    // ----------------------------------------------------------------------
    // Recirculate_Wash1:
    //  - Recirculates Wash 1 solvent to improve cleaning efficiency.
    // ----------------------------------------------------------------------
    E_WashingState.Recirculate_Wash1:

        RecirculateWash1();

        IF bMovementComplete THEN
            eWashingState    := E_WashingState.Cleaning_Lines_W1;
            iStepCounter     := 0;
            bMovementComplete := FALSE;
        END_IF


    // ----------------------------------------------------------------------
    // Cleaning_Lines_W1:
    //  - Cleans lines used for Wash 1 solvent.
    // ----------------------------------------------------------------------
    E_WashingState.Cleaning_Lines_W1:

        CleaningLinesWash1();

        IF bMovementComplete THEN
            eWashingState    := E_WashingState.Waste_Wash1;
            iStepCounter     := 0;
            bMovementComplete := FALSE;
        END_IF


    // ----------------------------------------------------------------------
    // Waste_Wash1:
    //  - Sends Wash 1 solvent remaining in lines to waste.
    //  - Then decides whether Wash 2 is enabled by recipe.
    // ----------------------------------------------------------------------
    E_WashingState.Waste_Wash1:

        WasteWash1();

        IF bMovementComplete THEN
            iStepCounter     := 0;
            bMovementComplete := FALSE;

            // Check if Wash 2 is active in the recipe:
            // aSolventN[4] > 0 → Wash 2 enabled
            IF GVL_Recipe.stActiveRecipe.stSolventsTimes.aSolventN[4] > 0 THEN
                eWashingState := E_WashingState.Metering_Wash2;
            ELSE
                eWashingState := E_WashingState.Completed;
            END_IF
        END_IF


    // ----------------------------------------------------------------------
    // Metering_Wash2:
    //  - Meters solvent for Wash 2 if configured in recipe.
    // ----------------------------------------------------------------------
    E_WashingState.Metering_Wash2:

        MeteringWash2();

        IF bMovementComplete THEN
            eWashingState    := E_WashingState.Recirculate_Wash2;
            iStepCounter     := 0;
            bMovementComplete := FALSE;
        END_IF


    // ----------------------------------------------------------------------
    // Recirculate_Wash2:
    //  - Recirculates Wash 2 solvent.
    // ----------------------------------------------------------------------
    E_WashingState.Recirculate_Wash2:

        RecirculateWash2();

        IF bMovementComplete THEN
            eWashingState    := E_WashingState.Cleaning_Lines_W2;
            iStepCounter     := 0;
            bMovementComplete := FALSE;
        END_IF


    // ----------------------------------------------------------------------
    // Cleaning_Lines_W2:
    //  - Cleans lines used for Wash 2 solvent.
    // ----------------------------------------------------------------------
    E_WashingState.Cleaning_Lines_W2:

        CleaningLinesWash2();

        IF bMovementComplete THEN
            eWashingState    := E_WashingState.Waste_Wash2;
            iStepCounter     := 0;
            bMovementComplete := FALSE;
        END_IF


    // ----------------------------------------------------------------------
    // Waste_Wash2:
    //  - Sends Wash 2 solvent remaining in lines to waste.
    // ----------------------------------------------------------------------
    E_WashingState.Waste_Wash2:

        WasteWash2();

        IF bMovementComplete THEN
            iStepCounter     := 0;
            bMovementComplete := FALSE;
            eWashingState    := E_WashingState.Completed;
        END_IF


    // ----------------------------------------------------------------------
    // Completed:
    //  - Washing phase has finished successfully.
    //  - Updates HMI and raises bWashingDone.
    // ----------------------------------------------------------------------
    E_WashingState.Completed:

        GVL_HMI.HMIAnimation.sLoadTextWashing   := 'Completed';
        GVL_HMI.HMIAnimation.rLoadBarWashing    := 100.0;
        GVL_HMI.HMIAnimation.eIconStateWashing  := E_IconState.Completed;

        bWashingDone  := TRUE;
        bWashingError := FALSE;


    // ----------------------------------------------------------------------
    // Error:
    //  - Generic washing error state (hook for future error handling).
    //  - Currently sets HMI to "Error" and raises bWashingError.
    // ----------------------------------------------------------------------
    E_WashingState.Error:

        GVL_HMI.HMIAnimation.sLoadTextWashing   := 'Error';
        GVL_HMI.HMIAnimation.rLoadBarWashing    := 0.0;
        GVL_HMI.HMIAnimation.eIconStateWashing  := E_IconState.Waiting;

        bWashingError := TRUE;
        bWashingDone  := FALSE;

END_CASE

ACTION CleaningLinesWash1:
//Exactly the oppisite of Recirculate Wash 1
CASE iStepCounter OF
	
	0: //Provide HMI animation details
		GVL_HMI.HMIAnimation.sLoadTextWashing := 'Cleaning Lines W1'; 
		iStepCounter := 1;
		
		FOR i := 1 TO 5 DO
			bMoveValveDone[i] := FALSE;
		END_FOR
		
    1: // Set valves on position 5 (Recirculating)
    	FOR i := 1 TO 5 DO
			IF NOT bMoveValveDone[i] THEN
			bMoveValveDone[i] := GVL_Motion.aValvesObj[i].MoveValve( iPosition := 5, 
																	 rVelocity := GVL_Motion.aValves[i].rTargetVel, 
																	 rAcc := GVL_Motion.aValves[i].rAcceleration, 
																	 rDec := GVL_Motion.aValves[i].rDeceleration 
																	);
			END_IF
		END_FOR
		
		IF bMoveValveDone[1] AND bMoveValveDone[2] AND bMoveValveDone[3] AND bMoveValveDone[4] AND bMoveValveDone[5] THEN
			FOR i := 1 TO 5 DO
				bMoveValveDone[i] := FALSE;
        	END_FOR
        	iStepCounter := 2;
		END_IF

    2: // Calculates the number of degrees of rotation of the pumps based on Wash 1 volume and factor 2

		fDistance[1] := F_VolumeToSteps(rVolume := (GVL_Recipe.stActiveRecipe.stVolumes.aT_IC_Volume[3] + GVL_Motion.aPumps[1].Rotary.rDeadVolume) * 2, iPumpIndex := 1);
		fDistance[2] := F_VolumeToSteps(rVolume := (GVL_Recipe.stActiveRecipe.stVolumes.aS0_Volume[3] + GVL_Motion.aPumps[2].Rotary.rDeadVolume) * 2, iPumpIndex := 2);
		fDistance[3] := F_VolumeToSteps(rVolume := (GVL_Recipe.stActiveRecipe.stVolumes.aS1_Volume[3] + GVL_Motion.aPumps[3].Rotary.rDeadVolume) * 2, iPumpIndex := 3);
		fDistance[4] := F_VolumeToSteps(rVolume := (GVL_Recipe.stActiveRecipe.stVolumes.aS2_Volume[3] + GVL_Motion.aPumps[4].Rotary.rDeadVolume) * 2, iPumpIndex := 4);
		fDistance[5] := F_VolumeToSteps(rVolume := (GVL_Recipe.stActiveRecipe.stVolumes.aS3_Volume[3] + GVL_Motion.aPumps[5].Rotary.rDeadVolume) * 2, iPumpIndex := 5);
		fDistance[6] := F_VolumeToSteps(rVolume := (GVL_Recipe.stActiveRecipe.stVolumes.aS4_Volume[3] + GVL_Motion.aPumps[6].Rotary.rDeadVolume) * 2, iPumpIndex := 6);
		fDistance[7] := F_VolumeToSteps(rVolume := (GVL_Recipe.stActiveRecipe.stVolumes.aS5_Volume[3] + GVL_Motion.aPumps[7].Rotary.rDeadVolume) * 2, iPumpIndex := 7);
		fDistance[8] := F_VolumeToSteps(rVolume := (GVL_Recipe.stActiveRecipe.stVolumes.aS6_Volume[3] + GVL_Motion.aPumps[8].Rotary.rDeadVolume) * 2, iPumpIndex := 8);
		fDistance[9] := F_VolumeToSteps(rVolume := (GVL_Recipe.stActiveRecipe.stVolumes.aS7_Volume[3] + GVL_Motion.aPumps[9].Rotary.rDeadVolume) * 2, iPumpIndex := 9);
		fDistance[10] := F_VolumeToSteps(rVolume := (GVL_Recipe.stActiveRecipe.stVolumes.aF_Volume[3] + GVL_Motion.aPumps[10].Rotary.rDeadVolume) * 2, iPumpIndex := 10);

		FOR i := 1 TO 10 DO
			bMovePumpDone[i] := FALSE;
		END_FOR
		
		iStepCounter := 3;
		
    3: // Starts rotary movement with calculated distance (degrees/sec -> steps) [positive movement]
        FOR i := 1 TO 10 DO
			IF NOT bMovePumpDone[i] THEN
				bMovePumpDone[i] := GVL_Motion.aPumpsRotary[i].MoveRelative( Distance := fDistance[i],
																			 Velocity := GVL_Settings.stPumpParameters.iRunVelocity * 6, 
																			 Acc := GVL_Settings.stPumpParameters.iRunVelocity * 3, 
																			 Dec := GVL_Settings.stPumpParameters.iRunVelocity * 3 
																			);
			END_IF
        END_FOR
		IF bMovePumpDone[1] AND bMovePumpDone[2] AND bMovePumpDone[3] AND bMovePumpDone[4] AND bMovePumpDone[5] AND bMovePumpDone[6] AND bMovePumpDone[7] AND bMovePumpDone[8] AND bMovePumpDone[9] AND bMovePumpDone[10] THEN
			FOR i := 1 TO 10 DO
				bMovePumpDone[i] := FALSE;
        	END_FOR
        	iStepCounter := 4; // Move to next step
		END_IF

    4: // Sets the movement done flag
		bMovementComplete := TRUE;
	
        
END_CASE
END_ACTION

ACTION CleaningLinesWash2:
//Exactly the oppisite of Recirculate Wash 1
CASE iStepCounter OF
	
	0: //Provide HMI animation details
		GVL_HMI.HMIAnimation.sLoadTextWashing := 'Cleaning Lines W2'; 
		iStepCounter := 1;
		
		FOR i := 1 TO 5 DO
			bMoveValveDone[i] := FALSE;
		END_FOR
		
    1: // Set valves on position 5 (Recirculating)
    	FOR i := 1 TO 5 DO
			IF NOT bMoveValveDone[i] THEN
			bMoveValveDone[i] := GVL_Motion.aValvesObj[i].MoveValve( iPosition := 5, 
																	 rVelocity := GVL_Motion.aValves[i].rTargetVel, 
																	 rAcc := GVL_Motion.aValves[i].rAcceleration, 
																	 rDec := GVL_Motion.aValves[i].rDeceleration 
																	);
			END_IF
		END_FOR
		
		IF bMoveValveDone[1] AND bMoveValveDone[2] AND bMoveValveDone[3] AND bMoveValveDone[4] AND bMoveValveDone[5] THEN
			FOR i := 1 TO 5 DO
				bMoveValveDone[i] := FALSE;
        	END_FOR
        	iStepCounter := 2;
		END_IF

    2: //Calculates the number of degrees of rotation of the pumps based on Wash 2 volume and factor 2

    	fDistance[1] := F_VolumeToSteps(rVolume := (GVL_Recipe.stActiveRecipe.stVolumes.aT_IC_Volume[4] + GVL_Motion.aPumps[1].Rotary.rDeadVolume) * 2, iPumpIndex := 1);
		fDistance[2] := F_VolumeToSteps(rVolume := (GVL_Recipe.stActiveRecipe.stVolumes.aS0_Volume[4] + GVL_Motion.aPumps[2].Rotary.rDeadVolume) * 2, iPumpIndex := 2);
		fDistance[3] := F_VolumeToSteps(rVolume := (GVL_Recipe.stActiveRecipe.stVolumes.aS1_Volume[4] + GVL_Motion.aPumps[3].Rotary.rDeadVolume) * 2, iPumpIndex := 3);
		fDistance[4] := F_VolumeToSteps(rVolume := (GVL_Recipe.stActiveRecipe.stVolumes.aS2_Volume[4] + GVL_Motion.aPumps[4].Rotary.rDeadVolume) * 2, iPumpIndex := 4);
		fDistance[5] := F_VolumeToSteps(rVolume := (GVL_Recipe.stActiveRecipe.stVolumes.aS3_Volume[4] + GVL_Motion.aPumps[5].Rotary.rDeadVolume) * 2, iPumpIndex := 5);
		fDistance[6] := F_VolumeToSteps(rVolume := (GVL_Recipe.stActiveRecipe.stVolumes.aS4_Volume[4] + GVL_Motion.aPumps[6].Rotary.rDeadVolume) * 2, iPumpIndex := 6);
		fDistance[7] := F_VolumeToSteps(rVolume := (GVL_Recipe.stActiveRecipe.stVolumes.aS5_Volume[4] + GVL_Motion.aPumps[7].Rotary.rDeadVolume) * 2, iPumpIndex := 7);
		fDistance[8] := F_VolumeToSteps(rVolume := (GVL_Recipe.stActiveRecipe.stVolumes.aS6_Volume[4] + GVL_Motion.aPumps[8].Rotary.rDeadVolume) * 2, iPumpIndex := 8);
		fDistance[9] := F_VolumeToSteps(rVolume := (GVL_Recipe.stActiveRecipe.stVolumes.aS7_Volume[4] + GVL_Motion.aPumps[9].Rotary.rDeadVolume) * 2, iPumpIndex := 9);
		fDistance[10] := F_VolumeToSteps(rVolume := (GVL_Recipe.stActiveRecipe.stVolumes.aF_Volume[4] + GVL_Motion.aPumps[10].Rotary.rDeadVolume) * 2, iPumpIndex := 10);

		FOR i := 1 TO 10 DO
			bMovePumpDone[i] := FALSE;
		END_FOR
		
		iStepCounter := 3;
		
    3: // Starts rotary movement with calculated distance (degrees/sec -> steps) [positive movement]
        FOR i := 1 TO 10 DO
			IF NOT bMovePumpDone[i] THEN
				bMovePumpDone[i] := GVL_Motion.aPumpsRotary[i].MoveRelative( Distance := fDistance[i],
																			 Velocity := GVL_Settings.stPumpParameters.iRunVelocity * 6, 
																			 Acc := GVL_Settings.stPumpParameters.iRunVelocity * 3, 
																			 Dec := GVL_Settings.stPumpParameters.iRunVelocity * 3 
																			);
			END_IF
        END_FOR
		IF bMovePumpDone[1] AND bMovePumpDone[2] AND bMovePumpDone[3] AND bMovePumpDone[4] AND bMovePumpDone[5] AND bMovePumpDone[6] AND bMovePumpDone[7] AND bMovePumpDone[8] AND bMovePumpDone[9] AND bMovePumpDone[10] THEN
			FOR i := 1 TO 10 DO
				bMovePumpDone[i] := FALSE;
        	END_FOR
        	iStepCounter := 4; // Move to next step
		END_IF

    4: // Sets the movement done flag
		bMovementComplete := TRUE;
	
        
END_CASE
END_ACTION

METHOD EstimateTotalTime : REAL
VAR
	i : INT;
    rTotalTime : REAL := 0.0;
    rTmpTime : REAL;
    rMaxPumpTime : REAL;
	aVolumesW1 : ARRAY[1..10] OF REAL;
	aVolumesW2 : ARRAY[1..10] OF REAL;
	rM2Travel : lREAL;
END_VAR
// --- Valve movements ---
// Estimated 1s per group of 5 valves per change (6 changes)
rTotalTime := rTotalTime + 1 * 6;

// --- Motor M2 movements --- (used in WasteWash1 and WasteWash2)
rM2Travel :=  ABS(GVL_Settings.stMachineParam.aM2Position[2] - GVL_Settings.stMachineParam.aM2Position[1]) / GVL_Settings.stMachineParam.rM2Velocity  //Waste Position Move
			+ ABS(GVL_Settings.stMachineParam.aM2Position[2] - GVL_Settings.stMachineParam.aM2Position[1]) / GVL_Settings.stMachineParam.rM2Velocity; //Home Position Move

rTotalTime := rTotalTime + rM2Travel * 2;

// --- Agitations (Recirculations) ---
rTotalTime := rTotalTime + TO_REAL(GVL_Recipe.stActiveRecipe.stOtherParams.tAgitate1Time) / 1000.0;
rTotalTime := rTotalTime + TO_REAL(GVL_Recipe.stActiveRecipe.stOtherParams.tAgitate2Time) / 1000.0;

// --- Pump phases executed in parallel ---
//Volume value tranfer Wash 1
aVolumesW1[1] := GVL_Recipe.stActiveRecipe.stVolumes.aT_IC_Volume[3];
aVolumesW1[2] := GVL_Recipe.stActiveRecipe.stVolumes.aS0_Volume[3];
aVolumesW1[3] := GVL_Recipe.stActiveRecipe.stVolumes.aS1_Volume[3];
aVolumesW1[4] := GVL_Recipe.stActiveRecipe.stVolumes.aS2_Volume[3];
aVolumesW1[5] := GVL_Recipe.stActiveRecipe.stVolumes.aS3_Volume[3];
aVolumesW1[6] := GVL_Recipe.stActiveRecipe.stVolumes.aS4_Volume[3];
aVolumesW1[7] := GVL_Recipe.stActiveRecipe.stVolumes.aS5_Volume[3];
aVolumesW1[8] := GVL_Recipe.stActiveRecipe.stVolumes.aS6_Volume[3];
aVolumesW1[9] := GVL_Recipe.stActiveRecipe.stVolumes.aS7_Volume[3];
aVolumesW1[10] := GVL_Recipe.stActiveRecipe.stVolumes.aF_Volume[3];
//Volume value tranfer Wash 2
aVolumesW2[1] := GVL_Recipe.stActiveRecipe.stVolumes.aT_IC_Volume[4];
aVolumesW2[2] := GVL_Recipe.stActiveRecipe.stVolumes.aS0_Volume[4];
aVolumesW2[3] := GVL_Recipe.stActiveRecipe.stVolumes.aS1_Volume[4];
aVolumesW2[4] := GVL_Recipe.stActiveRecipe.stVolumes.aS2_Volume[4];
aVolumesW2[5] := GVL_Recipe.stActiveRecipe.stVolumes.aS3_Volume[4];
aVolumesW2[6] := GVL_Recipe.stActiveRecipe.stVolumes.aS4_Volume[4];
aVolumesW2[7] := GVL_Recipe.stActiveRecipe.stVolumes.aS5_Volume[4];
aVolumesW2[8] := GVL_Recipe.stActiveRecipe.stVolumes.aS6_Volume[4];
aVolumesW2[9] := GVL_Recipe.stActiveRecipe.stVolumes.aS7_Volume[4];
aVolumesW2[10] := GVL_Recipe.stActiveRecipe.stVolumes.aF_Volume[4];

// For each block, use only the slowest pump
// MeteringWash1 (SolventN[3], Volumes[i][3])
IF GVL_Recipe.stActiveRecipe.stSolventsTimes.aSolventN[3] > 0 THEN
	rMaxPumpTime := 0;
	FOR i := 1 TO 10 DO
		rTmpTime := F_VolumeToSteps(rVolume := aVolumesW1[i], iPumpIndex := i) / GVL_Motion.aPumps[i].Rotary.rSpeed;
		IF rTmpTime > rMaxPumpTime THEN rMaxPumpTime := rTmpTime; END_IF
	END_FOR
	rTotalTime := rTotalTime + rMaxPumpTime;
END_IF

// MeteringWash2 (SolventN[4], Volumes[i][4])
IF GVL_Recipe.stActiveRecipe.stSolventsTimes.aSolventN[4] > 0 THEN
	rMaxPumpTime := 0;
	FOR i := 1 TO 10 DO
		rTmpTime := F_VolumeToSteps(rVolume := aVolumesW2[i], iPumpIndex := i) / GVL_Motion.aPumps[i].Rotary.rSpeed;
		IF rTmpTime > rMaxPumpTime THEN rMaxPumpTime := rTmpTime; END_IF
	END_FOR
	rTotalTime := rTotalTime + rMaxPumpTime;
END_IF

// WasteWash1 includes recipe volume + tubing dead volume (for each pump)
IF GVL_Recipe.stActiveRecipe.stSolventsTimes.aSolventN[3] > 0 THEN
	rMaxPumpTime := 0;
	FOR i := 1 TO 10 DO
		rTmpTime := F_VolumeToSteps(rVolume := aVolumesW1[i] + GVL_Motion.aPumps[i].Rotary.rDeadVolume, iPumpIndex := i) / GVL_Motion.aPumps[i].Rotary.rSpeed;
		IF rTmpTime > rMaxPumpTime THEN rMaxPumpTime := rTmpTime; END_IF
	END_FOR
	rTotalTime := rTotalTime + rMaxPumpTime;
END_IF

// WasteWash2 includes recipe volume + tubing dead volume (for each pump)
IF GVL_Recipe.stActiveRecipe.stSolventsTimes.aSolventN[4] > 0 THEN
	rMaxPumpTime := 0;
	FOR i := 1 TO 10 DO
		rTmpTime := F_VolumeToSteps(rVolume := aVolumesW2[i] + GVL_Motion.aPumps[i].Rotary.rDeadVolume, iPumpIndex := i) / GVL_Motion.aPumps[i].Rotary.rSpeed;
		IF rTmpTime > rMaxPumpTime THEN rMaxPumpTime := rTmpTime; END_IF
	END_FOR
	rTotalTime := rTotalTime + rMaxPumpTime;
END_IF

EstimateTotalTime := rTotalTime;
END_METHOD

ACTION MeteringWash1:
CASE iStepCounter OF
	
	0: //Provide HMI animation details
		GVL_HMI.HMIAnimation.sLoadTextWashing := 'Metering Wash 1'; 
		iStepCounter := 1; 
		FOR i := 1 TO 5 DO //reset valve movement flags
			bMoveValveDone[i] := FALSE;
		END_FOR
		
    1: // Set valves for Wash 1 position
	    FOR i := 1 TO 5 DO
			IF NOT bMoveValveDone[i] THEN
				bMoveValveDone[i] := GVL_Motion.aValvesObj[i].MoveValve(iPosition := GVL_Recipe.stActiveRecipe.stSolventsTimes.aSolventN[3], //Wash 1 solvent position
																	 	rVelocity := GVL_Motion.aValves[i].rTargetVel, 
																	 	rAcc := GVL_Motion.aValves[i].rAcceleration, 
																	 	rDec := GVL_Motion.aValves[i].rDeceleration 
																		);
			END_IF
			
        END_FOR
		
		IF bMoveValveDone[1] AND bMoveValveDone[2] AND bMoveValveDone[3] AND bMoveValveDone[4] AND bMoveValveDone[5] THEN
			FOR i := 1 TO 5 DO
				bMoveValveDone[i] := FALSE;
        	END_FOR
        	iStepCounter := 2;
		END_IF
        
	2: //Calculating the distance for each pump based on recipe volume plus tubing dead volume [Wash 1 - index 3]
		fDistance[1] := F_VolumeToSteps(rVolume := GVL_Recipe.stActiveRecipe.stVolumes.aT_IC_Volume[3] + GVL_Motion.aPumps[1].Rotary.rDeadVolume, iPumpIndex := 1);
		fDistance[2] := F_VolumeToSteps(rVolume := GVL_Recipe.stActiveRecipe.stVolumes.aS0_Volume[3] + GVL_Motion.aPumps[2].Rotary.rDeadVolume, iPumpIndex := 2);
		fDistance[3] := F_VolumeToSteps(rVolume := GVL_Recipe.stActiveRecipe.stVolumes.aS1_Volume[3] + GVL_Motion.aPumps[3].Rotary.rDeadVolume, iPumpIndex := 3);
		fDistance[4] := F_VolumeToSteps(rVolume := GVL_Recipe.stActiveRecipe.stVolumes.aS2_Volume[3] + GVL_Motion.aPumps[4].Rotary.rDeadVolume, iPumpIndex := 4);
		fDistance[5] := F_VolumeToSteps(rVolume := GVL_Recipe.stActiveRecipe.stVolumes.aS3_Volume[3] + GVL_Motion.aPumps[5].Rotary.rDeadVolume, iPumpIndex := 5);
		fDistance[6] := F_VolumeToSteps(rVolume := GVL_Recipe.stActiveRecipe.stVolumes.aS4_Volume[3] + GVL_Motion.aPumps[6].Rotary.rDeadVolume, iPumpIndex := 6);
		fDistance[7] := F_VolumeToSteps(rVolume := GVL_Recipe.stActiveRecipe.stVolumes.aS5_Volume[3] + GVL_Motion.aPumps[7].Rotary.rDeadVolume, iPumpIndex := 7);
		fDistance[8] := F_VolumeToSteps(rVolume := GVL_Recipe.stActiveRecipe.stVolumes.aS6_Volume[3] + GVL_Motion.aPumps[8].Rotary.rDeadVolume, iPumpIndex := 8);
		fDistance[9] := F_VolumeToSteps(rVolume := GVL_Recipe.stActiveRecipe.stVolumes.aS7_Volume[3] + GVL_Motion.aPumps[9].Rotary.rDeadVolume, iPumpIndex := 9);
		fDistance[10] := F_VolumeToSteps(rVolume := GVL_Recipe.stActiveRecipe.stVolumes.aF_Volume[3] + GVL_Motion.aPumps[10].Rotary.rDeadVolume, iPumpIndex := 10);
		
		FOR i := 1 TO 10 DO //reset pump movement flags
			bMovePumpDone[i] := FALSE;
		END_FOR
		
		iStepCounter := 3;
		
    3: // Performs rotary movement (positive movement)
        FOR i := 1 TO 10 DO
            IF NOT bMovePumpDone[i] THEN
				bMovePumpDone[i] := GVL_Motion.aPumpsRotary[i].MoveRelative( Distance := fDistance[i],
																			 Velocity := GVL_Settings.stPumpParameters.iMeterVelocity * 6,
																			 Acc := GVL_Settings.stPumpParameters.iMeterVelocity * 3, 
																			 Dec := GVL_Settings.stPumpParameters.iMeterVelocity * 3 
																			);
			END_IF
        END_FOR
		IF bMovePumpDone[1] AND bMovePumpDone[2] AND bMovePumpDone[3] AND bMovePumpDone[4] AND bMovePumpDone[5] AND bMovePumpDone[6] AND bMovePumpDone[7] AND bMovePumpDone[8] AND bMovePumpDone[9] AND bMovePumpDone[10] THEN
			FOR i := 1 TO 10 DO
				bMovePumpDone[i] := FALSE;
        	END_FOR
        	iStepCounter := 4; // Move to next step to monitor completion
		END_IF
	
	4: // Sets the movement done flag
		bMovementComplete := TRUE;
         
END_CASE
END_ACTION

ACTION MeteringWash2:
CASE iStepCounter OF
	
	0: //Provide HMI animation details
		GVL_HMI.HMIAnimation.sLoadTextWashing := 'Metering Wash 2'; 
		iStepCounter := 1; 
		FOR i := 1 TO 5 DO //reset valve movement flags
			bMoveValveDone[i] := FALSE;
		END_FOR
		
    1: // Set valves for Rinse 1 position
	    FOR i := 1 TO 5 DO
			IF NOT bMoveValveDone[i] THEN
				bMoveValveDone[i] := GVL_Motion.aValvesObj[i].MoveValve(iPosition := GVL_Recipe.stActiveRecipe.stSolventsTimes.aSolventN[4], //Wash 2 solvent position
																	 	rVelocity := GVL_Motion.aValves[i].rTargetVel, 
																	 	rAcc := GVL_Motion.aValves[i].rAcceleration, 
																	 	rDec := GVL_Motion.aValves[i].rDeceleration 
																		);
			END_IF
			
        END_FOR
		
		IF bMoveValveDone[1] AND bMoveValveDone[2] AND bMoveValveDone[3] AND bMoveValveDone[4] AND bMoveValveDone[5] THEN
			FOR i := 1 TO 5 DO
				bMoveValveDone[i] := FALSE;
        	END_FOR
        	iStepCounter := 2;
		END_IF
        
	2: //Calculating the distance for each pump based on recipe volume plus tubing dead volume [Wash 2 - index 4]
		fDistance[1] := F_VolumeToSteps(rVolume := GVL_Recipe.stActiveRecipe.stVolumes.aT_IC_Volume[4] + GVL_Motion.aPumps[1].Rotary.rDeadVolume, iPumpIndex := 1);
		fDistance[2] := F_VolumeToSteps(rVolume := GVL_Recipe.stActiveRecipe.stVolumes.aS0_Volume[4] + GVL_Motion.aPumps[2].Rotary.rDeadVolume, iPumpIndex := 2);
		fDistance[3] := F_VolumeToSteps(rVolume := GVL_Recipe.stActiveRecipe.stVolumes.aS1_Volume[4] + GVL_Motion.aPumps[3].Rotary.rDeadVolume, iPumpIndex := 3);
		fDistance[4] := F_VolumeToSteps(rVolume := GVL_Recipe.stActiveRecipe.stVolumes.aS2_Volume[4] + GVL_Motion.aPumps[4].Rotary.rDeadVolume, iPumpIndex := 4);
		fDistance[5] := F_VolumeToSteps(rVolume := GVL_Recipe.stActiveRecipe.stVolumes.aS3_Volume[4] + GVL_Motion.aPumps[5].Rotary.rDeadVolume, iPumpIndex := 5);
		fDistance[6] := F_VolumeToSteps(rVolume := GVL_Recipe.stActiveRecipe.stVolumes.aS4_Volume[4] + GVL_Motion.aPumps[6].Rotary.rDeadVolume, iPumpIndex := 6);
		fDistance[7] := F_VolumeToSteps(rVolume := GVL_Recipe.stActiveRecipe.stVolumes.aS5_Volume[4] + GVL_Motion.aPumps[7].Rotary.rDeadVolume, iPumpIndex := 7);
		fDistance[8] := F_VolumeToSteps(rVolume := GVL_Recipe.stActiveRecipe.stVolumes.aS6_Volume[4] + GVL_Motion.aPumps[8].Rotary.rDeadVolume, iPumpIndex := 8);
		fDistance[9] := F_VolumeToSteps(rVolume := GVL_Recipe.stActiveRecipe.stVolumes.aS7_Volume[4] + GVL_Motion.aPumps[9].Rotary.rDeadVolume, iPumpIndex := 9);
		fDistance[10] := F_VolumeToSteps(rVolume := GVL_Recipe.stActiveRecipe.stVolumes.aF_Volume[4] + GVL_Motion.aPumps[10].Rotary.rDeadVolume, iPumpIndex := 10);
		
		FOR i := 1 TO 10 DO //reset pump movement flags
			bMovePumpDone[i] := FALSE;
		END_FOR
		
		iStepCounter := 3;
		
    3: // Performs rotary movement (positive movement)
        FOR i := 1 TO 10 DO
            IF NOT bMovePumpDone[i] THEN
				bMovePumpDone[i] := GVL_Motion.aPumpsRotary[i].MoveRelative( Distance := fDistance[i],
																			 Velocity := GVL_Settings.stPumpParameters.iMeterVelocity * 6,
																			 Acc := GVL_Settings.stPumpParameters.iMeterVelocity * 3, 
																			 Dec := GVL_Settings.stPumpParameters.iMeterVelocity * 3 
																			);
			END_IF
        END_FOR
		IF bMovePumpDone[1] AND bMovePumpDone[2] AND bMovePumpDone[3] AND bMovePumpDone[4] AND bMovePumpDone[5] AND bMovePumpDone[6] AND bMovePumpDone[7] AND bMovePumpDone[8] AND bMovePumpDone[9] AND bMovePumpDone[10] THEN
			FOR i := 1 TO 10 DO
				bMovePumpDone[i] := FALSE;
        	END_FOR
        	iStepCounter := 4; // Move to next step to monitor completion
		END_IF
	
	4: // Sets the movement done flag
		bMovementComplete := TRUE;
         
END_CASE
END_ACTION

ACTION RecirculateWash1:
CASE iStepCounter OF
	
	0: //Provide HMI animation details
		GVL_HMI.HMIAnimation.sLoadTextWashing := 'Recirculate Wash 1'; 
		FOR i := 1 TO 5 DO
			bMoveValveDone[i] := FALSE;
		END_FOR
		iStepCounter := 1;
		
    1: // Set Valves position 5 (Recirculate)
    	FOR i := 1 TO 5 DO
			IF NOT bMoveValveDone[i] THEN
			bMoveValveDone[i] := GVL_Motion.aValvesObj[i].MoveValve( iPosition := 5, 
																	 rVelocity := GVL_Motion.aValves[i].rTargetVel, 
																	 rAcc := GVL_Motion.aValves[i].rAcceleration, 
																	 rDec := GVL_Motion.aValves[i].rDeceleration 
																	);
			END_IF
		END_FOR
		
		IF bMoveValveDone[1] AND bMoveValveDone[2] AND bMoveValveDone[3] AND bMoveValveDone[4] AND bMoveValveDone[5] THEN
			FOR i := 1 TO 5 DO
				bMoveValveDone[i] := FALSE;
        	END_FOR
        	iStepCounter := 2;
		END_IF

    2: // Calcula o numero de graus de rotacao das bombas baseado no tempo da receita Agitate Time 1

		fRecirculationTime  := TO_REAL(TIME_TO_DWORD(GVL_Recipe.stCurrentRecipe.stSolventsTimes.aTime[3])/1000);
		FOR i := 1 TO 10 DO
			fCalcDistance[i] 	:= fRecirculationTime * (GVL_Recipe.stActiveRecipe.stSolventsTimes.aVelocity[3] * 6);
		END_FOR
		
		FOR i := 1 TO 10 DO
			bMovePumpDone[i] := FALSE;
		END_FOR
		
		IF fRecirculationTime > 0 THEN
			iStepCounter := 3;
		END_IF
		
    3: // Inicia movimento rotativo com distância calculada (graus/seg -> steps) [negative moviment]
        FOR i := 1 TO 10 DO
			IF NOT bMovePumpDone[i] THEN
				bMovePumpDone[i] := GVL_Motion.aPumpsRotary[i].MoveRelative( Distance := - fCalcDistance[i],
																			 Velocity := GVL_Recipe.stActiveRecipe.stSolventsTimes.aVelocity[3] * 6, 
																			 Acc := GVL_Recipe.stActiveRecipe.stSolventsTimes.aVelocity[3] * 6, 
																			 Dec := GVL_Recipe.stActiveRecipe.stSolventsTimes.aVelocity[3] * 6 
																			);
			END_IF
        END_FOR
		IF bMovePumpDone[1] AND bMovePumpDone[2] AND bMovePumpDone[3] AND bMovePumpDone[4] AND bMovePumpDone[5] AND bMovePumpDone[6] AND bMovePumpDone[7] AND bMovePumpDone[8] AND bMovePumpDone[9] AND bMovePumpDone[10] THEN
			FOR i := 1 TO 10 DO
				bMovePumpDone[i] := FALSE;
        	END_FOR
        	iStepCounter := 4; // Move to next step to monitor completion
		END_IF

    4: // Sets the movement done flag
		bMovementComplete := TRUE;
	
        
END_CASE
END_ACTION

ACTION RecirculateWash2:
CASE iStepCounter OF
	
	0: //Provide HMI animation details
		GVL_HMI.HMIAnimation.sLoadTextWashing := 'Recirculate Wash 2'; 
		FOR i := 1 TO 5 DO
			bMoveValveDone[i] := FALSE;
		END_FOR
		iStepCounter := 1;
		
    1: // Set Valves position 5 (Recirculate)
    	FOR i := 1 TO 5 DO
			IF NOT bMoveValveDone[i] THEN
			bMoveValveDone[i] := GVL_Motion.aValvesObj[i].MoveValve( iPosition := 5, 
																	 rVelocity := GVL_Motion.aValves[i].rTargetVel, 
																	 rAcc := GVL_Motion.aValves[i].rAcceleration, 
																	 rDec := GVL_Motion.aValves[i].rDeceleration 
																	);
			END_IF
		END_FOR
		
		IF bMoveValveDone[1] AND bMoveValveDone[2] AND bMoveValveDone[3] AND bMoveValveDone[4] AND bMoveValveDone[5] THEN
			FOR i := 1 TO 5 DO
				bMoveValveDone[i] := FALSE;
        	END_FOR
        	iStepCounter := 2;
		END_IF

    2: // Calcula o numero de graus de rotacao das bombas baseado no tempo da receita Agitate Time 1

    	fRecirculationTime  := TO_REAL(TIME_TO_DWORD(GVL_Recipe.stCurrentRecipe.stSolventsTimes.aTime[4])/1000);
		FOR i := 1 TO 10 DO
			fCalcDistance[i] 	:= fRecirculationTime * (GVL_Recipe.stActiveRecipe.stSolventsTimes.aVelocity[4] * 6);
		END_FOR
		
		FOR i := 1 TO 10 DO
			bMovePumpDone[i] := FALSE;
		END_FOR
		
		IF fRecirculationTime > 0 THEN
			iStepCounter := 3;
		END_IF
		
    3: // Inicia movimento rotativo com distância calculada (graus/seg -> steps) [negative moviment]
        FOR i := 1 TO 10 DO
			IF NOT bMovePumpDone[i] THEN
				bMovePumpDone[i] := GVL_Motion.aPumpsRotary[i].MoveRelative( Distance := - fCalcDistance[i],
																			 Velocity := GVL_Recipe.stActiveRecipe.stSolventsTimes.aVelocity[4] * 6, 
																			 Acc := GVL_Recipe.stActiveRecipe.stSolventsTimes.aVelocity[4] * 6, 
																			 Dec := GVL_Recipe.stActiveRecipe.stSolventsTimes.aVelocity[4] * 6 
																			);
			END_IF
        END_FOR
		IF bMovePumpDone[1] AND bMovePumpDone[2] AND bMovePumpDone[3] AND bMovePumpDone[4] AND bMovePumpDone[5] AND bMovePumpDone[6] AND bMovePumpDone[7] AND bMovePumpDone[8] AND bMovePumpDone[9] AND bMovePumpDone[10] THEN
			FOR i := 1 TO 10 DO
				bMovePumpDone[i] := FALSE;
        	END_FOR
        	iStepCounter := 4; // Move to next step to monitor completion
		END_IF

    4: // Sets the movement done flag
		bMovementComplete := TRUE;
	
        
END_CASE
END_ACTION

METHOD Reset : BOOL
VAR_INPUT
END_VAR
//Init Flags
iStepCounter 	:= 0;
eWashingState := E_WashingState.Idle;

//Output flags
bWashingDone := FALSE;
bWashingError := FALSE;

// Control flags
iStepCounter := 0;
bStart := FALSE;
bMovementComplete := FALSE;

//Numbers variables
fAgitationTime    	:= 0.0;
fRecirculationTime	:= 0.0;
FOR i := 1 TO 10 DO
	fCalcDistance[i] := 0;
	fDistance[i] := 0;
END_FOR

//Movement Flags
bMoveM2 := FALSE;
FOR i := 1 TO 10 DO
	bMoveValveDone[i] := FALSE;
	bMovePumpDone[i] := FALSE;
END_FOR

//Icon progress reset
GVL_HMI.HMIAnimation.eIconStateWashing := E_IconState.Waiting;
GVL_HMI.HMIAnimation.rLoadBarWashing := 0;
tStartTime := T#0S;
rElapsedTimeSec := 0.0;
rTotalEstimatedTimeSec := 0.0;
bProgressInitDone := FALSE;

IF NOT bWashingDone AND NOT bWashingError THEN
	Reset := TRUE;
	RETURN;
ELSE
	Reset := FALSE;
END_IF
END_METHOD

ACTION WasteWash1:
CASE iStepCounter OF
	
	0: //Provide HMI animation details
		GVL_HMI.HMIAnimation.sLoadTextWashing := 'Waste Wash 1'; 
		
		FOR i := 1 TO 5 DO
			bMoveValveDone[i] := FALSE; // reset flags
		END_FOR
		
		iStepCounter := 1;
		
    1: // Set Valves into position 6 - Needles
    	FOR i := 1 TO 5 DO
			IF NOT bMoveValveDone[i] THEN
			bMoveValveDone[i] := GVL_Motion.aValvesObj[i].MoveValve( iPosition := 6, 
																	 rVelocity := GVL_Motion.aValves[i].rTargetVel, 
																	 rAcc := GVL_Motion.aValves[i].rAcceleration, 
																	 rDec := GVL_Motion.aValves[i].rDeceleration 
																	);
			END_IF
		END_FOR
		
		IF bMoveValveDone[1] AND bMoveValveDone[2] AND bMoveValveDone[3] AND bMoveValveDone[4] AND bMoveValveDone[5] THEN
			FOR i := 1 TO 5 DO
				bMoveValveDone[i] := FALSE; // reset flags
        	END_FOR
			bMoveM2 := FALSE;
        	iStepCounter := 2; //move to next step
		END_IF
		
	2: // M2 Motor movement
		IF NOT bMoveM2 THEN //Move M2 [Vertical Motor] to Waste position
			bMoveM2 := GVL_Motion.aMotors[2].MoveAbsolute(	rPosition := GVL_Settings.stMachineParam.aM2Position[2], 
															rVelocity := GVL_Settings.stMachineParam.rM2Velocity,
															rAcc := GVL_Settings.stMachineParam.rM2Accleration, 
															rDec := GVL_Settings.stMachineParam.rM2Deceleration	
														 	);
		END_IF
		
		// If M2 Movement is done, reset the flags and go to the next step
		IF bMoveM2  THEN
			bMoveM2 := FALSE;
			iStepCounter := 3;
		END_IF
		
    3: // Calculating distance for each pump
    	fDistance[1] := F_VolumeToSteps(rVolume := (GVL_Recipe.stActiveRecipe.stVolumes.aT_IC_Volume[3] + GVL_Motion.aPumps[1].Rotary.rDeadVolume) * 2.5 , iPumpIndex := 1);
		fDistance[2] := F_VolumeToSteps(rVolume := (GVL_Recipe.stActiveRecipe.stVolumes.aS0_Volume[3] + GVL_Motion.aPumps[2].Rotary.rDeadVolume) * 2.5, iPumpIndex := 2);
		fDistance[3] := F_VolumeToSteps(rVolume := (GVL_Recipe.stActiveRecipe.stVolumes.aS1_Volume[3] + GVL_Motion.aPumps[3].Rotary.rDeadVolume) * 2.5, iPumpIndex := 3);
		fDistance[4] := F_VolumeToSteps(rVolume := (GVL_Recipe.stActiveRecipe.stVolumes.aS2_Volume[3] + GVL_Motion.aPumps[4].Rotary.rDeadVolume) * 2.5, iPumpIndex := 4);
		fDistance[5] := F_VolumeToSteps(rVolume := (GVL_Recipe.stActiveRecipe.stVolumes.aS3_Volume[3] + GVL_Motion.aPumps[5].Rotary.rDeadVolume) * 2.5, iPumpIndex := 5);
		fDistance[6] := F_VolumeToSteps(rVolume := (GVL_Recipe.stActiveRecipe.stVolumes.aS4_Volume[3] + GVL_Motion.aPumps[6].Rotary.rDeadVolume) * 2.5, iPumpIndex := 6);
		fDistance[7] := F_VolumeToSteps(rVolume := (GVL_Recipe.stActiveRecipe.stVolumes.aS5_Volume[3] + GVL_Motion.aPumps[7].Rotary.rDeadVolume) * 2.5, iPumpIndex := 7);
		fDistance[8] := F_VolumeToSteps(rVolume := (GVL_Recipe.stActiveRecipe.stVolumes.aS6_Volume[3] + GVL_Motion.aPumps[8].Rotary.rDeadVolume) * 2.5, iPumpIndex := 8);
		fDistance[9] := F_VolumeToSteps(rVolume := (GVL_Recipe.stActiveRecipe.stVolumes.aS7_Volume[3] + GVL_Motion.aPumps[9].Rotary.rDeadVolume) * 2.5, iPumpIndex := 9);
		fDistance[10] := F_VolumeToSteps(rVolume := (GVL_Recipe.stActiveRecipe.stVolumes.aF_Volume[3] + GVL_Motion.aPumps[10].Rotary.rDeadVolume) * 2.5, iPumpIndex := 10);
		
		FOR i := 1 TO 10 DO
			bMovePumpDone[i] := FALSE; //resets pumps movement flags
		END_FOR
		
		iStepCounter := 4; // Move to next step
		
    4: // Start pumping by distance (degrees/seg -> steps) [negative moviment]
        FOR i := 1 TO 10 DO
			IF NOT bMovePumpDone[i] THEN
				bMovePumpDone[i] := GVL_Motion.aPumpsRotary[i].MoveRelative( Distance := - fDistance[i],
																			 Velocity := GVL_Settings.stPumpParameters.iRunVelocity * 6, 
																			 Acc := GVL_Settings.stPumpParameters.iRunVelocity * 6, 
																			 Dec := GVL_Settings.stPumpParameters.iRunVelocity * 6 
																			);
			END_IF
        END_FOR
		
		//Waits for every pump movement done flag
		IF bMovePumpDone[1] AND bMovePumpDone[2] AND bMovePumpDone[3] AND bMovePumpDone[4] AND bMovePumpDone[5] AND bMovePumpDone[6] AND bMovePumpDone[7] AND bMovePumpDone[8] AND bMovePumpDone[9] AND bMovePumpDone[10] THEN
			FOR i := 1 TO 10 DO
				bMovePumpDone[i] := FALSE;
        	END_FOR
        	iStepCounter := 5; // Move to next step
		END_IF

	5: //Resets M2 position
		IF NOT bMoveM2 THEN //Move M2 [Vertical Motor] to fill vials position after M3 movement is done
			bMoveM2 := GVL_Motion.aMotors[2].MoveAbsolute(	rPosition := GVL_Settings.stMachineParam.aM2Position[1], 
															rVelocity := GVL_Settings.stMachineParam.rM2Velocity,
															rAcc := GVL_Settings.stMachineParam.rM2Accleration, 
															rDec := GVL_Settings.stMachineParam.rM2Deceleration	
														 	);
		END_IF
		IF bMoveM2 THEN
			bMoveM2 := FALSE;
			iStepCounter := 6;
		END_IF
	
		
    6: // Sets the movement done flag
		bMovementComplete := TRUE;
	
        
END_CASE
END_ACTION

ACTION WasteWash2:
CASE iStepCounter OF
	
	0: //Provide HMI animation details
		GVL_HMI.HMIAnimation.sLoadTextWashing := 'Waste Wash 2'; 
		
		FOR i := 1 TO 5 DO
			bMoveValveDone[i] := FALSE; // reset flags
		END_FOR
		
		iStepCounter := 1;
		
    1: // Set Valves into position 6 - Needles
    	FOR i := 1 TO 5 DO
			IF NOT bMoveValveDone[i] THEN
			bMoveValveDone[i] := GVL_Motion.aValvesObj[i].MoveValve( iPosition := 6, 
																	 rVelocity := GVL_Motion.aValves[i].rTargetVel, 
																	 rAcc := GVL_Motion.aValves[i].rAcceleration, 
																	 rDec := GVL_Motion.aValves[i].rDeceleration 
																	);
			END_IF
		END_FOR
		
		IF bMoveValveDone[1] AND bMoveValveDone[2] AND bMoveValveDone[3] AND bMoveValveDone[4] AND bMoveValveDone[5] THEN
			FOR i := 1 TO 5 DO
				bMoveValveDone[i] := FALSE; // reset flags
        	END_FOR
			bMoveM2 := FALSE;
        	iStepCounter := 2; //move to next step
		END_IF
		
	2: // M2 Motor movement
		IF NOT bMoveM2 THEN //Move M2 [Vertical Motor] to Waste position
			bMoveM2 := GVL_Motion.aMotors[2].MoveAbsolute(	rPosition := GVL_Settings.stMachineParam.aM2Position[2], 
															rVelocity := GVL_Settings.stMachineParam.rM2Velocity,
															rAcc := GVL_Settings.stMachineParam.rM2Accleration, 
															rDec := GVL_Settings.stMachineParam.rM2Deceleration	
														 	);
		END_IF
		
		// If M2 Movement is done, reset the flags and go to the next step
		IF bMoveM2  THEN
			bMoveM2 := FALSE;
			iStepCounter := 3;
		END_IF
		
    3: // Calculating distance for each pump
    	fDistance[1] := F_VolumeToSteps(rVolume := (GVL_Recipe.stActiveRecipe.stVolumes.aT_IC_Volume[4] + GVL_Motion.aPumps[1].Rotary.rDeadVolume) * 2.5, iPumpIndex := 1);
		fDistance[2] := F_VolumeToSteps(rVolume := (GVL_Recipe.stActiveRecipe.stVolumes.aS0_Volume[4] + GVL_Motion.aPumps[2].Rotary.rDeadVolume) * 2.5, iPumpIndex := 2);
		fDistance[3] := F_VolumeToSteps(rVolume := (GVL_Recipe.stActiveRecipe.stVolumes.aS1_Volume[4] + GVL_Motion.aPumps[3].Rotary.rDeadVolume) * 2.5, iPumpIndex := 3);
		fDistance[4] := F_VolumeToSteps(rVolume := (GVL_Recipe.stActiveRecipe.stVolumes.aS2_Volume[4] + GVL_Motion.aPumps[4].Rotary.rDeadVolume) * 2.5, iPumpIndex := 4);
		fDistance[5] := F_VolumeToSteps(rVolume := (GVL_Recipe.stActiveRecipe.stVolumes.aS3_Volume[4] + GVL_Motion.aPumps[5].Rotary.rDeadVolume) * 2.5, iPumpIndex := 5);
		fDistance[6] := F_VolumeToSteps(rVolume := (GVL_Recipe.stActiveRecipe.stVolumes.aS4_Volume[4] + GVL_Motion.aPumps[6].Rotary.rDeadVolume) * 2.5, iPumpIndex := 6);
		fDistance[7] := F_VolumeToSteps(rVolume := (GVL_Recipe.stActiveRecipe.stVolumes.aS5_Volume[4] + GVL_Motion.aPumps[7].Rotary.rDeadVolume) * 2.5, iPumpIndex := 7);
		fDistance[8] := F_VolumeToSteps(rVolume := (GVL_Recipe.stActiveRecipe.stVolumes.aS6_Volume[4] + GVL_Motion.aPumps[8].Rotary.rDeadVolume) * 2.5, iPumpIndex := 8);
		fDistance[9] := F_VolumeToSteps(rVolume := (GVL_Recipe.stActiveRecipe.stVolumes.aS7_Volume[4] + GVL_Motion.aPumps[9].Rotary.rDeadVolume) * 2.5, iPumpIndex := 9);
		fDistance[10] := F_VolumeToSteps(rVolume := (GVL_Recipe.stActiveRecipe.stVolumes.aF_Volume[4] + GVL_Motion.aPumps[10].Rotary.rDeadVolume) * 2.5, iPumpIndex := 10);
		
		FOR i := 1 TO 10 DO
			bMovePumpDone[i] := FALSE; //resets pumps movement flags
		END_FOR
		
		iStepCounter := 4; // Move to next step
		
    4: // Start pumping by distance (degrees/seg -> steps) [negative moviment]
        FOR i := 1 TO 10 DO
			IF NOT bMovePumpDone[i] THEN
				bMovePumpDone[i] := GVL_Motion.aPumpsRotary[i].MoveRelative( Distance := - fDistance[i],
																			 Velocity := GVL_Settings.stPumpParameters.iRunVelocity * 6, 
																			 Acc := GVL_Settings.stPumpParameters.iRunVelocity * 6, 
																			 Dec := GVL_Settings.stPumpParameters.iRunVelocity * 6 
																			);
			END_IF
        END_FOR
		
		//Waits for every pump movement done flag
		IF bMovePumpDone[1] AND bMovePumpDone[2] AND bMovePumpDone[3] AND bMovePumpDone[4] AND bMovePumpDone[5] AND bMovePumpDone[6] AND bMovePumpDone[7] AND bMovePumpDone[8] AND bMovePumpDone[9] AND bMovePumpDone[10] THEN
			FOR i := 1 TO 10 DO
				bMovePumpDone[i] := FALSE;
        	END_FOR
        	iStepCounter := 5; // Move to next step
		END_IF

	5: //Resets M2 position
		IF NOT bMoveM2 THEN //Move M2 [Vertical Motor] to fill vials position after M3 movement is done
			bMoveM2 := GVL_Motion.aMotors[2].MoveAbsolute(	rPosition := GVL_Settings.stMachineParam.aM2Position[1], 
															rVelocity := GVL_Settings.stMachineParam.rM2Velocity,
															rAcc := GVL_Settings.stMachineParam.rM2Accleration, 
															rDec := GVL_Settings.stMachineParam.rM2Deceleration	
														 	);
		END_IF
		IF bMoveM2 THEN
			bMoveM2 := FALSE;
			iStepCounter := 6;
		END_IF
	
		
    6: // Sets the movement done flag
		bMovementComplete := TRUE;
	
        
END_CASE
END_ACTION

END_FUNCTION_BLOCK

// ---- POUs/2. AutoCycle/Stages/FB_DryingPhase.TcPOU
(*
    FB_DryingPhase
    ------------------------------------------------------------------------
    Purpose:
      - Orchestrates the full "Drying" macro-phase of the ASRS.
      - Sequence:
          1) Position M1 to the drying position (above Andersen stages)
          2) Open air supply through solenoids
          3) Maintain air flow for a configured drying time
          4) Close air supply and return solenoids to IDLE
          5) Move M1 back to the home position
          6) Mark phase as DONE

      - Updates HMI load bar and drying icon during the entire phase.

    Usage:
      - Call cyclically with bExecute = TRUE while the machine is in
        the Drying Phase state.
      - Internal state machine (eDryState) progresses through each step.
      - When eDryState reaches DONE and M1 is in home position,
        bDryingDone = TRUE.

    Inputs:
      - bExecute : BOOL
          TRUE  → start/continue the drying phase.
          FALSE → keeps FB in IDLE (no progression).

    Outputs:
      - bDryingDone  : BOOL
          TRUE when the drying sequence finished successfully.
      - bDryingError : BOOL
          TRUE if the phase enters ERROR state
          (currently a generic hook, no detailed error transitions here).

    Side Effects:
      - Writes to global HMI animation:
          GVL_HMI.HMIAnimation.eIconStateDry
          GVL_HMI.HMIAnimation.sLoadTextDry
          GVL_HMI.HMIAnimation.rLoadBarDry
      - Uses global motion/settings:
          GVL_Motion.M1Motor.rActualPos
          GVL_Motion.aMotors[1].MoveAbsolute(...)
          GVL_Settings.stMachineParam.aM1Position[1..2]
          GVL_Recipe.stActiveRecipe.stOtherParams.tAirDryTime
      - Uses solenoid control:
          GVL_IO.gSetSolenoidControl.PressureUp()
          GVL_IO.gSetSolenoidControl.Idle()
*)

FUNCTION_BLOCK FB_DryingPhase
VAR_INPUT
    bExecute : BOOL;  // TRUE to start/maintain drying phase
END_VAR

VAR_OUTPUT
    bDryingDone  : BOOL := FALSE; // TRUE when drying phase completes successfully
    bDryingError : BOOL := FALSE; // TRUE when an error occurs (ERROR state)
END_VAR

VAR
    // -----------------------------
    // Internal Drying FSM state
    // -----------------------------
    eDryState : (IDLE,          // Waiting for start
                 POSITION_M1,   // Move M1 to drying position
                 OPEN_AIR,      // Open air supply to stages
                 WAITING_TIME,  // Keep air on for configured time
                 CLOSE_AIR,     // Close air supply / return solenoids to idle
                 HOME_M1,       // Move M1 back to home position
                 DONE,          // Drying finished
                 ERROR);        // Error state

    // -----------------------------
    // Sub-function blocks
    // -----------------------------
    fbSolenoidControl : FB_SolenoidControl; // Solenoid control FB instance (not fully used here)
    tonAirDryTime     : TON;                // Timer to run air flow through stages

    // -----------------------------
    // Control flags
    // -----------------------------
    bStart          : BOOL := FALSE; // Start latch derived from bExecute
    bMoveM1         : BOOL := FALSE; // M1 vertical motor movement flag
    bM1RightPosition: BOOL := FALSE; // TRUE when M1 is within tolerance of target position

    // -----------------------------
    // HMI progress bar animation
    // -----------------------------
    tStartTime             : TIME := T#0S; // Drying start timestamp
    rElapsedTimeSec        : REAL := 0.0;  // Elapsed time in seconds
    rTotalEstimatedTimeSec : REAL := 0.0;  // Estimated total drying time (seconds)
    bProgressInitDone      : BOOL := FALSE; // Ensure estimation is done only once
END_VAR

(*
	* There is procedure doubts in here. Client says the drying phase leave stage closed and blow leak test pressure, around 4.2 psi. Now programmed this way.
	* Documentation says the stage should be opened and then blow main pressure, around 6 bar.
*)

// ==========================================================================
// 1) Start latch:
//    - On first bExecute = TRUE, latch bStart and initialize FSM to IDLE.
// ==========================================================================
IF NOT bStart THEN
    eDryState := IDLE;
    bStart    := bExecute;
END_IF

// ==========================================================================
// 2) HMI Progress Bar Animation
//    - Only updates while FSM is actively drying:
//        not IDLE, not DONE, not ERROR.
//    - Uses external EstimateTotalTime() to scale elapsed time into 0..100%.
// ==========================================================================
IF bProgressInitDone
   AND (eDryState <> IDLE)
   AND (eDryState <> DONE)
   AND (eDryState <> ERROR)
THEN
    // Elapsed time in seconds since drying started
    rElapsedTimeSec := TO_REAL(TIME() - tStartTime) / 100.0 / 10.0; // or /1000.0; adjust if needed
    // More explicit:
    // rElapsedTimeSec := TO_REAL(TIME() - tStartTime) / 1000.0;

    // Scale elapsed / estimated total into percentage
    GVL_HMI.HMIAnimation.rLoadBarDry :=
        MIN(100.0, rElapsedTimeSec / rTotalEstimatedTimeSec * 100.0);
END_IF

// ==========================================================================
// 3) Drying Phase FSM
// ==========================================================================
CASE eDryState OF

    // ----------------------------------------------------------------------
    // IDLE:
    //  - Reset flags and wait for bStart.
    //  - Initializes HMI and timing when phase starts.
    // ----------------------------------------------------------------------
    IDLE:

        // Reset outputs in Idle
        bDryingDone  := FALSE;
        bDryingError := FALSE;
        bMoveM1      := FALSE;

        IF bStart THEN
            // Initialize timing for drying progress
            tStartTime             := TIME();
            rTotalEstimatedTimeSec := EstimateTotalTime(); // External estimate
            bProgressInitDone      := TRUE;

            // Configure HMI animation for Drying Phase start
            GVL_HMI.HMIAnimation.eIconStateDry := E_IconState.InProgress;
            GVL_HMI.HMIAnimation.sLoadTextDry  := 'Starting';
            GVL_HMI.HMIAnimation.rLoadBarDry   := 0.0;

            // Move to first step: position M1 for drying
            eDryState := POSITION_M1;
        END_IF


    // ----------------------------------------------------------------------
    // POSITION_M1:
    //  - Move M1 to the drying position (above Andersen stages).
    // ----------------------------------------------------------------------
    POSITION_M1:

        // Update HMI text
        GVL_HMI.HMIAnimation.sLoadTextDry := 'Moving Motor';

        // Start movement to drying position if not already triggered
        IF NOT bMoveM1 THEN
            bMoveM1 := GVL_Motion.aMotors[1].MoveAbsolute(
                rPosition := GVL_Settings.stMachineParam.aM1Position[2],
                rVelocity := GVL_Settings.stMachineParam.rM1Velocity,
                rAcc      := GVL_Settings.stMachineParam.rM1Accleration,
                rDec      := GVL_Settings.stMachineParam.rM1Deceleration
            );
        END_IF

        // When MoveAbsolute reports TRUE (command accepted/completed depending on wrapper),
        // go to next step to open air
        IF bMoveM1 THEN
            bMoveM1   := FALSE;          // Reset movement flag for next moves
            eDryState := OPEN_AIR;       // Next step
        END_IF


    // ----------------------------------------------------------------------
    // OPEN_AIR:
    //  - Ensure M1 is in the right position and then open air supply
    //    using solenoid control.
	// ----------------------------------------------------------------------
    OPEN_AIR:

        // Check if M1 is at the drying position within tolerance
        bM1RightPosition :=
            ABS(GVL_Motion.M1Motor.rActualPos - GVL_Settings.stMachineParam.aM1Position[2]) <= 2.0;

        IF bM1RightPosition THEN
            // Raise pressure via solenoid control (air ON)
            IF GVL_IO.gSetSolenoidControl.PressureUp() THEN
                eDryState := WAITING_TIME; // Next: wait for configured air drying time
            END_IF
        ELSE
            // If position is not correct, go back to POSITION_M1
            bMoveM1   := FALSE;
            eDryState := POSITION_M1;
        END_IF


    // ----------------------------------------------------------------------
    // WAITING_TIME:
    //  - Keep air flowing for the configured drying time (tAirDryTime).
    // ----------------------------------------------------------------------
    WAITING_TIME:

        // Update HMI text
        GVL_HMI.HMIAnimation.sLoadTextDry := 'Drying';

        // Start/maintain timer for air drying time
        tonAirDryTime(
            IN := TRUE,
            PT := GVL_Recipe.stActiveRecipe.stOtherParams.tAirDryTime
        );

        // When timer completes, go to close air step
        IF tonAirDryTime.Q THEN
            eDryState := CLOSE_AIR;
        END_IF


    // ----------------------------------------------------------------------
    // CLOSE_AIR:
    //  - Turn off air supply and return solenoids to idle.
// ----------------------------------------------------------------------
    CLOSE_AIR:

        // Reset timer input
        tonAirDryTime(IN := FALSE);

        // Set solenoids to idle position (air OFF, safe position)
        IF GVL_IO.gSetSolenoidControl.Idle() THEN
            bMoveM1   := FALSE;
            eDryState := HOME_M1; // Next: move M1 back home
        END_IF


    // ----------------------------------------------------------------------
    // HOME_M1:
    //  - Move M1 back to home position after drying.
    // ----------------------------------------------------------------------
    HOME_M1:

        // Update HMI text
        GVL_HMI.HMIAnimation.sLoadTextDry := 'Homing Motor';

        // Command M1 to home/initial position if not already triggered
        IF NOT bMoveM1 THEN
            bMoveM1 := GVL_Motion.aMotors[1].MoveAbsolute(
                rPosition := GVL_Settings.stMachineParam.aM1Position[1],
                rVelocity := GVL_Settings.stMachineParam.rM1Velocity,
                rAcc      := GVL_Settings.stMachineParam.rM1Accleration,
                rDec      := GVL_Settings.stMachineParam.rM1Deceleration
            );
        END_IF

        // When movement is finished, go to DONE state
        IF bMoveM1 THEN
            bMoveM1   := FALSE;
            eDryState := DONE;
        END_IF


    // ----------------------------------------------------------------------
    // DONE:
    //  - Final state when drying phase is completed successfully.
    //  - Validates M1 position and updates HMI + done flag.
    // ----------------------------------------------------------------------
    DONE:

        // Confirm that M1 is at home position within tolerance
        bM1RightPosition :=
            ABS(GVL_Motion.M1Motor.rActualPos - GVL_Settings.stMachineParam.aM1Position[1]) <= 2.0;

        IF bM1RightPosition THEN
            // HMI animation: drying completed
            GVL_HMI.HMIAnimation.eIconStateDry := E_IconState.Completed;
            GVL_HMI.HMIAnimation.sLoadTextDry  := 'Completed';
            GVL_HMI.HMIAnimation.rLoadBarDry   := 100.0;

            // Success flag
            bDryingDone  := TRUE;
            bDryingError := FALSE;
        ELSE
            // If position is not correct, try to home again
            bMoveM1   := FALSE;
            eDryState := HOME_M1;
        END_IF


    // ----------------------------------------------------------------------
    // ERROR:
    //  - Generic drying error state (hook for future detailed handling).
    //  - Currently only updates HMI and sets bDryingError.
    // ----------------------------------------------------------------------
    ERROR:

        // HMI animation: error state
        GVL_HMI.HMIAnimation.sLoadTextDry   := 'Error';
        GVL_HMI.HMIAnimation.rLoadBarDry    := 0.0;
        GVL_HMI.HMIAnimation.eIconStateDry  := E_IconState.Waiting;

        bDryingError := TRUE;
        bDryingDone  := FALSE;

END_CASE

METHOD EstimateTotalTime : REAL
VAR
	rTotalTime : LREAL := 0.0;
    rDistance : LREAL;
    rVelocity : LREAL;
END_VAR
// --- Motor M1 movement (sequential) ---
rDistance := ABS(GVL_Settings.stMachineParam.aM1Position[2] - GVL_Settings.stMachineParam.aM1Position[3]); //From seal position up to dry position
rVelocity := GVL_Settings.stMachineParam.rM1Velocity;
IF rVelocity > 0 THEN
    rTotalTime := rTotalTime + rDistance / rVelocity;
END_IF

// --- Solenoid switching times (estimated 0.5s per switch) ---
rTotalTime := rTotalTime + 0.5 * 3; // open_air, close_air, reset

// --- Timer duration from recipe (AirDryTime) ---
rTotalTime := rTotalTime + TO_REAL(GVL_Recipe.stActiveRecipe.stOtherParams.tAirDryTime) / 1000.0;

EstimateTotalTime := rTotalTime;
END_METHOD

METHOD Reset : BOOL
VAR_INPUT
END_VAR
//output flags
bDryingDone  := FALSE;
bDryingError  := FALSE;

//state machine sequence
eDryState	:= IDLE;

//fb's and timers
//fbSolenoidControl(bExecute := FALSE);
tonAirDryTime(In := FALSE);

//initiation flags
bStart := FALSE; 
bMoveM1 := FALSE; 

//Progress bar variables
tStartTime := T#0S;
rElapsedTimeSec := 0.0;
rTotalEstimatedTimeSec := 0.0;
bProgressInitDone := FALSE;
GVL_HMI.HMIAnimation.rLoadBarDry := 0;

IF NOT bDryingDone AND NOT bDryingError THEN
	Reset := TRUE;
	RETURN;
ELSE
	Reset := FALSE;
END_IF
END_METHOD

END_FUNCTION_BLOCK

// ---- POUs/2. AutoCycle/Stages/FB_SealStages.TcPOU
(*
    FB_SealStages
    ----------------------------------------
    Purpose:
      - Execute the "sealing" movement of Motor M1 to a predefined position.
      - Uses a two-step positioning strategy:
          1) Fast move to a pre-position (with deceleration offset)
          2) Precise move to the final seal position
      - Provides status back to the caller (bSealSuccess / bSealError).
      - Updates HMI animation (text, icon state and progress bar).

    Usage:
      - Call with bExecute = TRUE cyclically while the auto cycle is in
        the sealing step.
      - bSealSuccess becomes TRUE when M1 reaches the target position
        within tolerance.
      - bSealError becomes TRUE if a motion error is detected.
*)

FUNCTION_BLOCK FB_SealStages
VAR_INPUT
    bExecute : BOOL;   // TRUE to start/maintain the sealing sequence
END_VAR

VAR_OUTPUT
    bSealSuccess : BOOL; // TRUE when sealing sequence completes successfully
    bSealError   : BOOL; // TRUE if an error occurs during execution
END_VAR

VAR
    // -----------------------------
    // Execution & positioning
    // -----------------------------
    bExecuting      : BOOL := FALSE; // TRUE after first cycle with bExecute = TRUE
    rActualPosition : LREAL;         // Current position of M1
    rTargetPosition : LREAL;         // Final sealing position for M1
    rTolerance      : LREAL := 0.5;  // Allowed position tolerance for "in position"
    bInPosition     : BOOL := FALSE; // TRUE when |actual - target| <= tolerance

    // Two-step motion sequence flags
    bMoveM1Pos1 : BOOL := FALSE;     // TRUE when pre-position move is completed
    bMoveM1Pos2 : BOOL := FALSE;     // TRUE when final precision move is completed

    bMotionSequenceDone : BOOL := FALSE; // TRUE when both steps are completed

    // Timer and trigger for second move
    bStartMove2  : BOOL := FALSE;    // Internal trigger to start second move
    tonStartMove2: TON;              // Timer between move 1 and move 2

    stStatus : ST_ActuatorStatus;    // Status structure returned by motor wrapper

    // -----------------------------
    // HMI Icon / Progress Bar
    // -----------------------------
    rElapsedTimeSec : REAL := 0.0;   // Elapsed time since FB start (seconds)
    tStartTime      : TIME := T#0S;  // Time when execution started
    bLoadBarUpdate  : BOOL := FALSE; // TRUE while progress bar should be updated
END_VAR

// ==========================================================================
// 1) Read actual position and evaluate "in position"
// ==========================================================================
rActualPosition := GVL_Motion.M1Motor.rActualPos;                     // Read current motor position
rTargetPosition := GVL_Settings.stMachineParam.aM1Position[2];        // Sealing target position (index 2)
bInPosition     := ABS(rActualPosition - rTargetPosition) <= rTolerance;

// ==========================================================================
// 2) HMI: basic sealing animation state
// ==========================================================================
GVL_HMI.HMIAnimation.sLoadTextSealing   := 'Sealing';
GVL_HMI.HMIAnimation.eIconStateSealing := E_IconState.InProgress;

// ==========================================================================
// 3) HMI: Load bar update (only while executing and not yet in position)
//    - Uses an external function EstimateTotalTime() to estimate total
//      sealing time, and scales elapsed time into 0..100%.
// ==========================================================================
IF bExecuting AND NOT bInPosition THEN
    // Elapsed time in seconds since FB start
    rElapsedTimeSec := TIME_TO_REAL(TIME() - tStartTime) / 1000.0;

    // Protect against division by zero or invalid estimate
    IF EstimateTotalTime() > 0.0 THEN
        GVL_HMI.HMIAnimation.rLoadBarSealing :=
            LIMIT(0.0,
                  (rElapsedTimeSec / EstimateTotalTime()) * 100.0,
                  100.0);
    ELSE
        GVL_HMI.HMIAnimation.rLoadBarSealing := 0.0;
    END_IF
END_IF

// ==========================================================================
// 4) Main execution logic: only runs when bExecute = TRUE
// ==========================================================================
IF bExecute THEN

    // -------------------------------------------------------------
    // 4.1) First entry initialization (rising edge of bExecute)
    //      - Reset internal flags and start timing for the load bar
    // -------------------------------------------------------------
    IF NOT bExecuting THEN
        bExecuting      := TRUE;
        bLoadBarUpdate  := TRUE;

        bMoveM1Pos1     := FALSE;
        bMoveM1Pos2     := FALSE;
        bStartMove2     := FALSE;
        bMotionSequenceDone := FALSE;

        tStartTime      := TIME();       // Reference start time
        tonStartMove2(IN := FALSE);      // Reset timer input

        // Reset progress bar only once at the beginning
        GVL_HMI.HMIAnimation.rLoadBarSealing := 0.0;
    END_IF

    // -------------------------------------------------------------
    // 4.2) Execute two-step motion sequence while:
    //      - M1 is not yet in final position, or
    //      - the motion sequence is not finished
    // -------------------------------------------------------------
    IF NOT bInPosition OR NOT bMotionSequenceDone THEN

        // If both moves are completed, flag sequence as done
        IF bMoveM1Pos1 AND bMoveM1Pos2 THEN
            bStartMove2        := FALSE;
            bMotionSequenceDone := TRUE;
        END_IF

        // ---------------------------------------------------------
        // Step 1: Move M1 to a pre-position (with deceleration offset)
        //         This allows a faster approach before the precision step.
        // ---------------------------------------------------------
        IF NOT bMoveM1Pos1 THEN
            bMoveM1Pos1 := GVL_Motion.aMotors[1].MoveAbsolute(
                rPosition := rTargetPosition + GVL_Settings.stMachineParam.fM1PositionDeceleration,
                rVelocity := GVL_Settings.stMachineParam.rM1Velocity,
                rAcc      := GVL_Settings.stMachineParam.rM1Accleration,
                rDec      := GVL_Settings.stMachineParam.rM1Deceleration
            );
        END_IF

        // When step 1 is completed, start the trigger for step 2
        IF bMoveM1Pos1 AND NOT bMoveM1Pos2 THEN
            bStartMove2 := TRUE;
        END_IF

        // Timer between step 1 and step 2 (settling time)
        tonStartMove2(IN := bStartMove2, PT := T#500MS);

        // ---------------------------------------------------------
        // Step 2: Final precise move to the exact target position
        //         - Uses a lower velocity for better accuracy.
        // ---------------------------------------------------------
        IF NOT bMoveM1Pos2 AND tonStartMove2.Q THEN
            bMoveM1Pos2 := GVL_Motion.aMotors[1].MoveAbsolute(
                rPosition := rTargetPosition,
                rVelocity := GVL_Settings.stMachineParam.rM1PrecisionVelocity,
                rAcc      := GVL_Settings.stMachineParam.rM1Accleration,
                rDec      := GVL_Settings.stMachineParam.rM1Deceleration
            );
        END_IF
    END_IF

    // -------------------------------------------------------------
    // 4.3) Read motor status and evaluate error / success
    // -------------------------------------------------------------
    stStatus := GVL_Motion.aMotors[1].GetStatus();

    // --- Error handling ---
    IF stStatus.bError THEN
        bSealError   := TRUE;
        bSealSuccess := FALSE;

    ELSE
        bSealError := FALSE;

        // --- Success condition: M1 is within target tolerance ---
        IF bInPosition THEN
            bSealSuccess  := TRUE;
            bLoadBarUpdate := FALSE;

            // Force progress bar and HMI icon to "Completed"
            GVL_HMI.HMIAnimation.rLoadBarSealing   := 100.0;
            GVL_HMI.HMIAnimation.eIconStateSealing := E_IconState.Completed;
        ELSE
            bSealSuccess := FALSE;
        END_IF
    END_IF

END_IF

METHOD EstimateTotalTime : REAL
VAR
	rDist1      : LREAL;   // Distance for Move 1 (pre-position with deceleration offset)
    rDist2      : LREAL;   // Distance for Move 2 (final precision move)
    rVel1       : LREAL;   // Velocity for Move 1
    rVel2       : LREAL;   // Velocity for Move 2
    rTimeMove1  : REAL;    // Estimated time for Move 1
    rTimeMove2  : REAL;    // Estimated time for Move 2
END_VAR
// Move 1: from actual position → target + decel offset
rDist1 := ABS(
    (GVL_Settings.stMachineParam.aM1Position[2] +
     GVL_Settings.stMachineParam.fM1PositionDeceleration)
    - GVL_Motion.M1Motor.rActualPos
);

// Move 2: from pre-position → final target
rDist2 := ABS(
    GVL_Settings.stMachineParam.aM1Position[2] -
    (GVL_Settings.stMachineParam.aM1Position[2] +
     GVL_Settings.stMachineParam.fM1PositionDeceleration)
);

// ----------------------------------------------------------
// READ VELOCITIES FOR EACH MOVEMENT
// ----------------------------------------------------------
rVel1 := GVL_Settings.stMachineParam.rM1Velocity;           // Fast move
rVel2 := GVL_Settings.stMachineParam.rM1PrecisionVelocity;  // Precision move

// ----------------------------------------------------------
// ESTIMATE DURATIONS (simple distance / velocity)
// ----------------------------------------------------------

// Estimated time for Move 1
IF rVel1 > 0 THEN
    rTimeMove1 := rDist1 / rVel1 * 1.5;
END_IF

// Estimated time for Move 2
IF rVel2 > 0 THEN
    rTimeMove2 := rDist2 / rVel2 * 1.5;
END_IF

// ----------------------------------------------------------
// FINAL CALCULATION
// Total time = Move 1 + 500 ms delay + Move 2
// ----------------------------------------------------------
EstimateTotalTime := rTimeMove1 + 0.5 + rTimeMove2 + 15;
END_METHOD

METHOD Reset : BOOL
VAR_INPUT
END_VAR
// Reset Flags
bSealSuccess	:= FALSE;
bSealError  	:= FALSE;
bInPosition		:= FALSE;
bMotionSequenceDone	:= FALSE;	


bExecuting		:= FALSE;
rActualPosition	:= 0.0;
rTargetPosition := 0.0;
bMoveM1Pos1	 	:= FALSE;
bMoveM1Pos2	 	:= FALSE;
bStartMove2		:= FALSE;
tonStartMove2( IN := FALSE);

rElapsedTimeSec := 0.0;
tStartTime 		:= T#0S;
bLoadBarUpdate 	:= FALSE;

// Send Reset Return
IF NOT bSealSuccess AND NOT bSealError THEN
	Reset := TRUE;
	RETURN;
ELSE
	Reset := FALSE;
END_IF
END_METHOD

END_FUNCTION_BLOCK

// ---- POUs/2. AutoCycle/Stages/FB_LeakTest.TcPOU
(*
==============================================================================
 FB_LeakTest
------------------------------------------------------------------------------
 Purpose:
   - Perform an automatic leak test on the Andersen / ASRS system.
   - Sequence:
       1) Move all 6-position valves to leak test position (pos. 6).
       2) Optionally seal stages by moving M1 to the sealing position.
       3) Set solenoids to "PressureUp" and build pressure for a defined time.
       4) Close air and hold pressure.
       5) Monitor the pressure over a configured time window.
       6) Pass criteria: measured pressure >= configured threshold.
       7) If pressure drops below threshold → test fails (ERROR).

 HMI:
   - The action ACT_LoadingIcon handles:
       * Animation of the leak test progress bar.
       * Estimation of the total leak test duration.
   - This FB updates:
       * GVL_HMI.HMIAnimation.sLoadTextLeakTest
       * GVL_HMI.HMIAnimation.rLoadBarLeakTest
       * GVL_HMI.HMIAnimation.eIconStateLeakTest

 Usage:
   - Call cyclically with:
        bExecute := TRUE
        eSolenoidPosition := E_SolenoidSet.LEAKTEST (from AutoCycle)
        tPressureUpTime   := <seconds>
        tMonitorTime      := <seconds>
   - Outputs:
        bLeakTestDone  = TRUE  → leak test passed.
        bLeakTestError = TRUE  → leak test failed or valve error.
        rSystemPressure        → current scaled pressure (PSI).
        sLTMessageError        → error description (on failure).
   - Call Reset() to clear internal state before a new leak test.
==============================================================================
*)

FUNCTION_BLOCK FB_LeakTest
VAR_INPUT
    bExecute          : BOOL;       // Start command for leak test
    eSolenoidPosition : E_SolenoidSet; // Solenoid configuration (not used directly here)
    tMonitorTime      : UINT;       // Monitoring duration [s]
    tPressureUpTime   : UINT;       // Pressurization duration [s]
END_VAR

VAR_OUTPUT
    bLeakTestDone   : BOOL;                 // TRUE when leak test finished successfully
    rSystemPressure : LREAL;                // Current scaled system pressure (PSI)
    bLeakTestError  : BOOL;                 // TRUE if any error or failure during leak test
    sLTMessageError : STRING(100);          // Human readable description of leak test failure
END_VAR

VAR
    // Valve and solenoid / sensor helper blocks
    aValveMoveDone  : ARRAY[1..5] OF BOOL;  // TRUE when each valve finishes moving
    fbSolenoidControl : FB_SolenoidControl; // Not directly used here (we call gSetSolenoidControl)
    fbSensorScaling : FB_SensorScaling;     // Reserved for future scaling use

    // Pressure / timing flags
    bPressureInput  : BOOL := FALSE;        // Internal enable for monitoring TON
    tStartTime      : TIME;                 // Reserved (not used in current implementation)
    rScaledPressure : REAL;                 // Raw scaled pressure in PSI
    eState          : (IDLE, POSITION_VALVES, SET_SOLENOIDS, SEAL_STAGES, PRESSURIZE, CLOSE_AIR, MONITOR, RELEASE_AIR, DONE, ERROR); //Implicit_Enum__FB_LeakTest__eState; // Internal state machine

    bMoveValves        : BOOL := FALSE;     // Internal "valve move" flag
    bPressureTime      : BOOL := FALSE;     // Enables pressurization TON
    bPressureTaken     : BOOL := FALSE;     // TRUE when pressure threshold is captured
    bMoveM1MotorFast   : BOOL := FALSE;     // Fast movement part of M1 sealing (coarse position)
    bMoveM1MotorSlow   : BOOL := FALSE;     // Slow, precise movement of M1 to sealing position
    bM1MoveStartDelay  : BOOL := FALSE;     // Delay between fast and slow M1 movements
	bLeakTestPassed	   : BOOL := FALSE;     // Leak test passed flag
	
    rClosedSystemPressure : REAL := 0.0;    // Pressure threshold limit (from settings)

    // Timers
    tonPressuring   : TON;                  // Timer for pressure build-up phase
    tonMonitoring   : TON;                  // Timer for pressure monitoring phase
    tonM1MoveDelay  : TON;                  // Delay between fast and slow M1 moves
    tonIconLoading  : TON;                  // Progress bar animation timer

    tLoadingTotalTime : TIME;               // Total time used by ACT_LoadingIcon
    bLoadTimeTaken    : BOOL := FALSE;      // TRUE once total time is calculated

    // Actuator status and debug
    stStatus      : ARRAY[1..5] OF ST_ActuatorStatus; // Status of each valve
    i             : USINT := 0;                        // Generic loop index
    fbEventHandler : FB_EventHandler;                  // Event logger instance
    bExecuteEvent : BOOL := FALSE;                     // Trigger for event logger
    bEventDone    : BOOL := FALSE;                     // Event logger completion

    rTargetPosition : INT;                             // Reserved (not used currently)
    bIconAnimation  : BOOL;                            // TRUE when leak-test load bar is active

    bDebug : ARRAY[1..10] OF BOOL;                    // Debug flags (for online analysis)
END_VAR

//=============================================================================
// Main body
//=============================================================================

// 1) HMI icon animation and load-bar handling (time estimation)
ACT_LoadingIcon();

ACT_CalScreenStatus();

// 2) Leak-test state machine
CASE eState OF

    //=====================================================================
    // IDLE
    //  - Waiting for bExecute to start a new leak test.
    //=====================================================================
    IDLE:
        // Start only if requested and there is no pending DONE / ERROR
        IF bExecute AND NOT (bLeakTestDone OR bLeakTestError) THEN
            // Initialize HMI animation
            GVL_HMI.HMIAnimation.sLoadTextLeakTest  := 'Starting';
            GVL_HMI.HMIAnimation.rLoadBarLeakTest   := 0.0;
            GVL_HMI.HMIAnimation.eIconStateLeakTest := E_IconState.InProgress;

            // Reset timing flags for new run
            bLoadTimeTaken := FALSE;
            tonMonitoring(IN := FALSE);
            tonPressuring(IN := FALSE);

            // Move to first step: valve positioning
            eState := POSITION_VALVES;
        END_IF;


    //=====================================================================
    // POSITION_VALVES
    //  - Move all 6-position valves to position 6 (LeakTest configuration).
    //  - Decide whether we need to seal stages (M1 movement) before pressure.
    //=====================================================================
    POSITION_VALVES:
        // Update HMI text
        GVL_HMI.HMIAnimation.sLoadTextLeakTest := 'Positioning Valves';
        bMoveValves := bExecute; // currently not used directly, but kept for clarity

        // Move all valves to position 6 (LeakTest / Needles)
        IF NOT aValveMoveDone[1] THEN
            aValveMoveDone[1] := GVL_Motion.aValvesObj[1].MoveValve(
                iPosition := 6,
                rVelocity := GVL_Motion.aValves[1].rTargetVel,
                rAcc      := GVL_Motion.aValves[1].rAcceleration,
                rDec      := GVL_Motion.aValves[1].rDeceleration
            );
        END_IF

        IF NOT aValveMoveDone[2] THEN
            aValveMoveDone[2] := GVL_Motion.aValvesObj[2].MoveValve(
                iPosition := 6,
                rVelocity := GVL_Motion.aValves[2].rTargetVel,
                rAcc      := GVL_Motion.aValves[2].rAcceleration,
                rDec      := GVL_Motion.aValves[2].rDeceleration
            );
        END_IF

        IF NOT aValveMoveDone[3] THEN
            aValveMoveDone[3] := GVL_Motion.aValvesObj[3].MoveValve(
                iPosition := 6,
                rVelocity := GVL_Motion.aValves[3].rTargetVel,
                rAcc      := GVL_Motion.aValves[3].rAcceleration,
                rDec      := GVL_Motion.aValves[3].rDeceleration
            );
        END_IF

        IF NOT aValveMoveDone[4] THEN
            aValveMoveDone[4] := GVL_Motion.aValvesObj[4].MoveValve(
                iPosition := 6,
                rVelocity := GVL_Motion.aValves[4].rTargetVel,
                rAcc      := GVL_Motion.aValves[4].rAcceleration,
                rDec      := GVL_Motion.aValves[4].rDeceleration
            );
        END_IF

        IF NOT aValveMoveDone[5] THEN
            aValveMoveDone[5] := GVL_Motion.aValvesObj[5].MoveValve(
                iPosition := 6,
                rVelocity := GVL_Motion.aValves[5].rTargetVel,
                rAcc      := GVL_Motion.aValves[5].rAcceleration,
                rDec      := GVL_Motion.aValves[5].rDeceleration
            );
        END_IF

        // Read status of each valve actuator
        stStatus[1] := GVL_Motion.aValvesObj[1].GetStatus();
        stStatus[2] := GVL_Motion.aValvesObj[2].GetStatus();
        stStatus[3] := GVL_Motion.aValvesObj[3].GetStatus();
        stStatus[4] := GVL_Motion.aValvesObj[4].GetStatus();
        stStatus[5] := GVL_Motion.aValvesObj[5].GetStatus();

        // All valves in position 6 → continue
        IF    aValveMoveDone[1]
           AND aValveMoveDone[2]
           AND aValveMoveDone[3]
           AND aValveMoveDone[4]
           AND aValveMoveDone[5] THEN

            bMoveValves := FALSE;

            // Decide whether we must re-seal stages (M1 position check)
            IF GVL_Motion.M1Motor.rActualPos <= (GVL_Settings.stMachineParam.aM1Position[2] + 0.5) THEN
                // Already at or very close to sealing position, set solenoids
                eState := SET_SOLENOIDS;
            ELSE
                // Need to move M1 through the sealing sequence first
                eState := SEAL_STAGES;
            END_IF

            // Reset valve move flags for next use
            FOR i := 1 TO 5 DO
                aValveMoveDone[i] := FALSE;
            END_FOR
        END_IF

        // If any valve reports an error → leak test error
        IF    stStatus[1].bError
           OR stStatus[2].bError
           OR stStatus[3].bError
           OR stStatus[4].bError
           OR stStatus[5].bError THEN

            bLeakTestError  := TRUE;
            sLTMessageError := 'Failed to position valves';

            eState := ERROR;
        END_IF;


    //=====================================================================
    // SEAL_STAGES
    //  - 2-step motion of M1 to the sealing position:
    //      1) Fast move to an offset near target.
    //      2) Delayed slow move to precise sealing position.
    //=====================================================================
    SEAL_STAGES:
        // Delay between fast and slow movement
        tonM1MoveDelay(IN := bM1MoveStartDelay, PT := T#500MS);

        // Start delay once fast move is triggered
        IF bMoveM1MotorFast THEN
            bM1MoveStartDelay := TRUE;
        END_IF

        // Step 1: fast move close to target (with deceleration offset)
        IF NOT bMoveM1MotorFast THEN
            bMoveM1MotorFast := GVL_Motion.aMotors[1].MoveAbsolute(
                rPosition := GVL_Settings.stMachineParam.aM1Position[2] + GVL_Settings.stMachineParam.fM1PositionDeceleration,
                rVelocity := GVL_Settings.stMachineParam.rM1Velocity,
                rAcc      := GVL_Settings.stMachineParam.rM1Accleration,
                rDec      := GVL_Settings.stMachineParam.rM1Deceleration
            );
        END_IF

        // Step 2: precise slow move to sealing position (after delay)
        IF NOT bMoveM1MotorSlow AND bMoveM1MotorFast AND tonM1MoveDelay.Q THEN
            bMoveM1MotorSlow := GVL_Motion.aMotors[1].MoveAbsolute(
                rPosition := GVL_Settings.stMachineParam.aM1Position[2],
                rVelocity := GVL_Settings.stMachineParam.rM1PrecisionVelocity,
                rAcc      := GVL_Settings.stMachineParam.rM1Accleration,
                rDec      := GVL_Settings.stMachineParam.rM1Deceleration
            );
        END_IF

        // Both steps completed → clear flags and proceed to solenoids
        IF bMoveM1MotorSlow AND bMoveM1MotorFast THEN
            tonM1MoveDelay(IN := FALSE, PT := T#500MS);
            bM1MoveStartDelay := FALSE;

            bMoveM1MotorSlow := FALSE;
            bMoveM1MotorFast := FALSE;

            eState := SET_SOLENOIDS;
        END_IF


    //=====================================================================
    // SET_SOLENOIDS
    //  - Set solenoids to "PressureUp" configuration to start pressurization.
    //=====================================================================
    SET_SOLENOIDS:
        // Request solenoid group to go to "PressureUp" (air in)
        IF GVL_IO.gSetSolenoidControl.PressureUp() THEN
            bPressureTime := TRUE;
            eState        := PRESSURIZE;
        END_IF


    //=====================================================================
    // PRESSURIZE
    //  - Build pressure for tPressureUpTime seconds.
    //=====================================================================
    PRESSURIZE:
        // Update HMI text
        GVL_HMI.HMIAnimation.sLoadTextLeakTest := 'Pressurizing';

        // Run pressurization timer (tPressureUpTime is in seconds)
        tonPressuring(
            IN := bPressureTime,
            PT := UINT_TO_TIME(tPressureUpTime * 1000)
        );

        IF tonPressuring.Q THEN
            // Stop pressure timing and close air path
            bPressureTime := FALSE;
            eState        := CLOSE_AIR;
        END_IF;


    //=====================================================================
    // CLOSE_AIR
    //  - Switch solenoids to "HoldPressure" to create a closed system for
    //    monitoring.
    //=====================================================================
    CLOSE_AIR:
        // Set the solenoids to "HoldPressure" configuration
        IF GVL_IO.gSetSolenoidControl.HoldPressure() THEN
            bPressureTime := TRUE;
            eState        := MONITOR;
        END_IF


    //=====================================================================
    // MONITOR
    //  - Monitor the leak test pressure over the configured time window.
    //  - If pressure stays above threshold until timer expires → DONE.
    //  - If pressure drops below the threshold at any time → ERROR.
    //=====================================================================
    MONITOR:
        // Update HMI text
        GVL_HMI.HMIAnimation.sLoadTextLeakTest := 'Monitoring';

        // Scale raw sensor input to PSI
        //   NOTE: Calibration based on 4–20 mA range:
        //         220 .. 6100 = 0 .. 3.698 V (example) → PSI
        rScaledPressure :=
            (GVL_IO.gAnalogInputs.rLeakTestPressureSensor - 220.0)
            * (3.698 / (6100.0 - 220.0));

        // First pass: capture the allowed leak-test pressure limit
        IF NOT bPressureTaken THEN
            rClosedSystemPressure := GVL_Settings.stLeakTestParameters.rLeakTestPressureLimit;
            bPressureTaken        := TRUE;
            bPressureInput        := TRUE;  // enable monitoring timer
        ELSE
            // Run monitoring timer (tMonitorTime is in seconds)
            tonMonitoring(
                IN := bPressureInput,
                PT := UDINT_TO_TIME(tMonitorTime * 1000)
            );

            // Check pressure criteria
            IF (rScaledPressure >= rClosedSystemPressure) AND tonMonitoring.Q THEN
                // Pressure stayed above limit during full monitoring window
                bPressureTaken := FALSE;
				bLeakTestPassed := TRUE;
                eState         := RELEASE_AIR;

            ELSIF rScaledPressure < rClosedSystemPressure THEN
                // Pressure dropped below limit before timer expired
                bPressureTaken := FALSE;
				bLeakTestPassed := FALSE;
                eState         := RELEASE_AIR;
            END_IF
        END_IF

        // Export pressure for HMI and external monitoring
        GVL_HMI.rCalLeakTestPressure := rScaledPressure;
        rSystemPressure              := rScaledPressure;

		
	 //=====================================================================
    // RELEASE_AIR
    //  - Release the air inside the system.
    //=====================================================================
    RELEASE_AIR:
		// Set the solenoids to "Idle" configuration
        IF GVL_IO.gSetSolenoidControl.Idle() THEN
            IF bLeakTestPassed THEN
				eState        := DONE;
			ELSE
				eState        := ERROR;
			END_IF
        END_IF
		

    //=====================================================================
    // DONE
    //  - Leak test successfully completed and HMI is updated accordingly.
    //  - Wait for bExecute to go FALSE to return to IDLE for next run.
    //=====================================================================
    DONE:
		// HMI final state for successful leak test if on auto cycle state
		IF (GVL_HMI.eMachineMode = E_MachineMode.AUTO_CYCLE) THEN
			GVL_HMI.HMIAnimation.rLoadBarLeakTest   := 100.0;
			GVL_HMI.HMIAnimation.sLoadTextLeakTest  := 'Completed';
			GVL_HMI.HMIAnimation.eIconStateLeakTest := E_IconState.Completed;
		END_IF
        
        bLeakTestDone := TRUE;

        // Wait for start command to be released before going back to IDLE
        IF NOT bExecute THEN
            eState        := IDLE;
            bLeakTestDone := FALSE;
        END_IF


    //=====================================================================
    // ERROR
    //  - Leak test failed or an error occurred.
    //  - bLeakTestError must be checked by caller.
    //  - Wait for bExecute to go FALSE to return to IDLE.
    //=====================================================================
    ERROR:
        bLeakTestError := TRUE;
        // HMI: error is indicated by load bar / text via ACT_LoadingIcon and
        //      external handling of sLTMessageError.

        IF NOT bExecute THEN
            eState        := IDLE;
            bLeakTestDone := FALSE;
        END_IF

END_CASE;

ACTION ACT_CalScreenStatus:
IF GVL_HMI.bCalLeakTestButton THEN
	CASE eState OF
	
		POSITION_VALVES:
			GVL_HMI.sCalLeakTestStatus := 'Idle';
			GVL_HMI.iCalLeakTestState  := 1;
		
		PRESSURIZE:
			GVL_HMI.sCalLeakTestStatus := 'Pressuring up';
			GVL_HMI.iCalLeakTestState  := 1;
		
		MONITOR:
			GVL_HMI.sCalLeakTestStatus := 'Monitoring';
			GVL_HMI.iCalLeakTestState  := 1;
		
		DONE:
			GVL_HMI.sCalLeakTestStatus := 'Passed';
			GVL_HMI.iCalLeakTestState  := 2;
		
		ERROR:
			GVL_HMI.sCalLeakTestStatus := 'Failed';
			GVL_HMI.iCalLeakTestState  := 3;
			
	END_CASE	
END_IF
END_ACTION

ACTION ACT_LoadingIcon:
(*
==============================================================================
 ACT_LoadingIcon
------------------------------------------------------------------------------
 Purpose:
   - Compute a rough estimated time for the leak test (pressurize + monitor).
   - Drive the HMI leak-test progress bar (rLoadBarLeakTest) based on a TON.
   - Only active in AUTO_CYCLE mode; otherwise, the bar is reset to 0%.

 Behaviour:
   - When machine mode is AUTO_CYCLE:
       1) On first activation, calculate tLoadingTotalTime:
             (tPressureUpTime + tMonitorTime) seconds + 500 ms margin.
       2) Run tonIconLoading for that total duration.
       3) HMI bar = (ET / TotalTime) * 100.
   - When not in AUTO_CYCLE:
       - Reset timer, flags and bar.
==============================================================================
*)

// Decide if we should animate the icon based on machine mode
IF GVL_HMI.eMachineMode = E_MachineMode.AUTO_CYCLE THEN
    bIconAnimation := TRUE;
ELSE
    bIconAnimation := FALSE;
END_IF

IF bIconAnimation THEN

    // Compute total estimated time only once per leak-test execution
    IF NOT bLoadTimeTaken THEN
        // tPressureUpTime and tMonitorTime in seconds → convert to TIME in ms
        tLoadingTotalTime :=
            UINT_TO_TIME((tPressureUpTime * 1000) + (tMonitorTime * 1000) + 500);
        bLoadTimeTaken := TRUE;
    END_IF

    // Run TON that will be used as base for the HMI bar
    tonIconLoading(
        IN := bIconAnimation,
        PT := tLoadingTotalTime
    );

    // Protect against division by zero
    IF tLoadingTotalTime > T#0MS THEN
        // Progress bar = (ET / TotalTime) * 100
        GVL_HMI.HMIAnimation.rLoadBarLeakTest :=
            (TIME_TO_REAL(tonIconLoading.ET) * 100.0) / TIME_TO_REAL(tLoadingTotalTime);
    ELSE
        GVL_HMI.HMIAnimation.rLoadBarLeakTest := 0.0;
    END_IF

ELSE
    // When animation is disabled (e.g., not in AUTO_CYCLE):
    // - Stop timer
    // - Clear flag so it will be recalculated next time
    // - Reset HMI bar
    tonIconLoading(IN := FALSE);
    bLoadTimeTaken := FALSE;
    GVL_HMI.HMIAnimation.rLoadBarLeakTest := 0.0;
END_IF
END_ACTION

(*
==============================================================================
 Method: Reset
------------------------------------------------------------------------------
 Purpose:
   - Reset FB_LeakTest internal state and HMI outputs so a new leak test
     can start cleanly.
   - This method does NOT automatically restart the test; the caller must
     set bExecute := TRUE again to run a new cycle.

 Behaviour:
   - Clears:
       * Valve flags, pressure flags, timers, internal state (eState).
       * HMI leak-test icon state (set to Waiting).
       * Outputs related to current run (pressure and error text).
   - Returns:
       Reset = TRUE  when the block is ready for a new start
                     (bLeakTestDone = FALSE and bLeakTestError = FALSE).
       Reset = FALSE otherwise.
==============================================================================
*)
METHOD Reset : BOOL
VAR
    i : USINT;
END_VAR
// Reset per-valve movement flags
FOR i := 1 TO 5 DO
    aValveMoveDone[i] := FALSE;
END_FOR

// Reset pressure-related flags and outputs
bPressureInput   := FALSE;
bPressureTime    := FALSE;
bPressureTaken   := FALSE;
bExecuteEvent    := FALSE;
bEventDone       := FALSE;
bLeakTestError   := FALSE;
bLoadTimeTaken   := FALSE;
bLeakTestDone    := FALSE;
rSystemPressure  := 0.0;
sLTMessageError  := '';
rScaledPressure  := 0.0;

// Reset internal state and motion flags
eState             := IDLE;
bMoveValves        := FALSE;
bMoveM1MotorFast   := FALSE;
bMoveM1MotorSlow   := FALSE;
bM1MoveStartDelay  := FALSE;
rClosedSystemPressure := 0.0;

// Reset timers
tonPressuring(IN := FALSE);
tonMonitoring(IN := FALSE);
tonM1MoveDelay(IN := FALSE);
tonIconLoading(IN := FALSE);

tLoadingTotalTime := T#0S;
rTargetPosition   := 1;
bIconAnimation    := FALSE;

// Reset leak test icon to "Waiting" state in HMI
GVL_HMI.HMIAnimation.eIconStateLeakTest := E_IconState.Waiting;

// Return TRUE only if no DONE or ERROR is currently active
IF NOT bLeakTestDone AND NOT bLeakTestError THEN
    Reset := TRUE;
    RETURN;
ELSE
    Reset := FALSE;
END_IF
END_METHOD

END_FUNCTION_BLOCK

// ---- POUs/2. AutoCycle/Stages/FB_PrimeSolvent.TcPOU
(*
==============================================================================
 FB_PrimeSolvent
------------------------------------------------------------------------------
 Purpose:
   - Automatically prime only the solvents that are actually used in the
     active recipe (Rinse1, Rinse2, Wash1, Wash2).
   - For each solvent that appears in the recipe (1..4), perform a generic
     prime cycle:
        1) Set valves to solvent position (1..4)
        2) Pump forward (from bottle towards jars) to fill lines
        3) Set valves to needles position (6)
        4) Pump backward (from jars to waste) to empty jars and keep lines full
   - Provides an HMI progress bar and status text for the priming phase.

 Usage:
   - Call cyclically with bExecute := TRUE to start.
   - Monitor:
        bDone  = TRUE  → prime sequence finished
        bError = TRUE  → reserved for future validation / error handling
   - After bDone, call Reset() before starting a new prime sequence.
==============================================================================
*)
FUNCTION_BLOCK FB_PrimeSolvent
VAR_INPUT
    bExecute : BOOL;  // Start command for the prime sequence (edge-detected)
END_VAR

VAR_OUTPUT
    bDone  : BOOL;    // Prime sequence completed successfully
    bError : BOOL;    // Reserved for future validation / error handling
END_VAR

VAR
    // Prime state machine control
    ePrimeState : E_PrimeSolventState := E_PrimeSolventState.PS_Idle;  // Main prime FSM state
    bStart      : BOOL := FALSE;                                       // Latches rising edge of bExecute
    bBusy       : BOOL := FALSE;                                       // Indicates this FB is currently running

    // Internal step machine for a single solvent prime cycle
    iStepCounter      : INT  := 0;     // Generic step counter used by PrimeSolventCycle()
    bMovementComplete : BOOL := FALSE; // TRUE when the current solvent cycle is finished

    // Motion flags for valves and pumps
    bMoveValveDone : ARRAY[1..5] OF BOOL := [FALSE, FALSE, FALSE, FALSE, FALSE];  // Per-valve completion flags
    bMovePumpDone  : ARRAY[1..10] OF BOOL := [FALSE, FALSE, FALSE, FALSE, FALSE,
                                              FALSE, FALSE, FALSE, FALSE, FALSE]; // Per-pump completion flags

    // Pump distances (steps) for each rotary pump
    fDistance : ARRAY[1..10] OF REAL;  // Steps to move each pump, computed from volume via F_VolumeToSteps()

    // Prime volumes (in ml)
    rPrimeForwardVolume  : REAL := 35.0;   // Forward prime volume (bottle → jars/lines)
    rPrimeBackwardVolume : REAL := 100.0;  // Backward prime volume (jars → waste, keep lines primed)

    // Solvent selection based on recipe
    iActiveSolventPosition : USINT := 0;   // Current solvent position being primed (1..4 = valve positions)
    bPrimeRequired         : ARRAY[1..4] OF BOOL := [FALSE, FALSE, FALSE, FALSE];
                                           // TRUE if that solvent (1..4) must be primed according to recipe
    iNumSolventsToPrime    : INT := 0;     // Number of unique solvents that actually need priming

    // Loop helpers
    iSolventIdx : INT;  // index for scanning solvents 1..4
    iStage      : INT;  // index for scanning recipe stages (Rinse1..Wash2)
    iSolventNum : INT;  // solvent number read from recipe (0..4)
    i           : INT;  // generic loop index

    // HMI progress bar support
    tStartTime             : TIME;     // Timestamp when prime sequence started
    rElapsedTimeSec        : REAL;     // Elapsed time since start, in seconds
    rTotalEstimatedTimeSec : REAL := 60.0;  // Estimated total prime duration (s). Overwritten by EstimateTotalTime()
    bProgressInitDone      : BOOL := FALSE; // Ensures estimation and HMI init is done only once
END_VAR

//=============================================================================
// Main body
//=============================================================================

IF NOT bStart THEN
    // First scan: initialise internal state and latch start condition
    ePrimeState := E_PrimeSolventState.PS_Idle;
    bStart      := bExecute;  // rising edge detection simplified (bExecute must go FALSE before next start)
END_IF

// --------------------------------------------------------------------------
// Progress bar handling
//   - Active only while prime is running (not IDLE or COMPLETED).
//   - Uses elapsed time / estimated total time to compute %.
// --------------------------------------------------------------------------
IF bProgressInitDone
   AND (ePrimeState <> E_PrimeSolventState.PS_Idle)
   AND (ePrimeState <> E_PrimeSolventState.PS_Completed) THEN

    // Compute elapsed time in seconds
    rElapsedTimeSec := TO_REAL(TIME() - tStartTime) / 1000.0;

    // Protect HMI bar from going over 100%
    GVL_HMI.HMIAnimation.rLoadBarPrime :=
        MIN(100.0, rElapsedTimeSec / rTotalEstimatedTimeSec * 100.0);
END_IF


// --------------------------------------------------------------------------
// Prime state machine
// --------------------------------------------------------------------------
CASE ePrimeState OF

    //=====================================================================
    // IDLE
    //  - Wait here until bStart is latched (bExecute rising edge).
    //  - Builds prime list from recipe and either:
    //       * finishes immediately if nothing to prime, or
    //       * moves to solvent 1 state to start the sequence.
    //=====================================================================
    E_PrimeSolventState.PS_Idle:

        // Reset public and internal flags
        bDone  := FALSE;
        bError := FALSE;
        bBusy  := FALSE;

        IF bStart THEN
            // Build list of which solvents (1..4) are actually used in recipe
            BuildPrimeListFromRecipe();

            IF iNumSolventsToPrime = 0 THEN
                // No prime required: directly complete phase
                GVL_HMI.HMIAnimation.sLoadTextPrime  := 'Prime skipped';
                GVL_HMI.HMIAnimation.rLoadBarPrime   := 100.0;
                GVL_HMI.HMIAnimation.eIconStatePrime := E_IconState.Completed;

                bDone       := TRUE;
                ePrimeState := E_PrimeSolventState.PS_Completed;
            ELSE
                // Configure progress bar timing and HMI texts
                tStartTime             := TIME();
                rTotalEstimatedTimeSec := EstimateTotalTime();
                bProgressInitDone      := TRUE;

                GVL_HMI.HMIAnimation.sLoadTextPrime  := 'Prime Solvents';
                GVL_HMI.HMIAnimation.rLoadBarPrime   := 0.0;
                GVL_HMI.HMIAnimation.eIconStatePrime := E_IconState.InProgress;

                // Start from solvent 1
                ePrimeState       := E_PrimeSolventState.PS_Solvent1;
                iStepCounter      := 0;
                bMovementComplete := FALSE;
                bBusy             := TRUE;
            END_IF
        END_IF


    //=====================================================================
    // PRIME SOLVENT 1 (valve position 1)
    //  - Skip if not required by recipe.
    //  - Otherwise run generic prime cycle with iActiveSolventPosition = 1.
    //=====================================================================
    E_PrimeSolventState.PS_Solvent1:

        IF NOT bPrimeRequired[1] THEN
            // Solvent 1 not used → skip to next solvent
            ePrimeState       := E_PrimeSolventState.PS_Solvent2;
            iStepCounter      := 0;
            bMovementComplete := FALSE;
        ELSE
            iActiveSolventPosition := 1;
            PrimeSolventCycle();  // uses iStepCounter internally

            IF bMovementComplete THEN
                // Move to solvent 2
                ePrimeState       := E_PrimeSolventState.PS_Solvent2;
                iStepCounter      := 0;
                bMovementComplete := FALSE;
            END_IF
        END_IF


    //=====================================================================
    // PRIME SOLVENT 2 (valve position 2)
    //=====================================================================
    E_PrimeSolventState.PS_Solvent2:

        IF NOT bPrimeRequired[2] THEN
            ePrimeState       := E_PrimeSolventState.PS_Solvent3;
            iStepCounter      := 0;
            bMovementComplete := FALSE;
        ELSE
            iActiveSolventPosition := 2;
            PrimeSolventCycle();

            IF bMovementComplete THEN
                ePrimeState       := E_PrimeSolventState.PS_Solvent3;
                iStepCounter      := 0;
                bMovementComplete := FALSE;
            END_IF
        END_IF


    //=====================================================================
    // PRIME SOLVENT 3 (valve position 3)
    //=====================================================================
    E_PrimeSolventState.PS_Solvent3:

        IF NOT bPrimeRequired[3] THEN
            ePrimeState       := E_PrimeSolventState.PS_Solvent4;
            iStepCounter      := 0;
            bMovementComplete := FALSE;
        ELSE
            iActiveSolventPosition := 3;
            PrimeSolventCycle();

            IF bMovementComplete THEN
                ePrimeState       := E_PrimeSolventState.PS_Solvent4;
                iStepCounter      := 0;
                bMovementComplete := FALSE;
            END_IF
        END_IF


    //=====================================================================
    // PRIME SOLVENT 4 (valve position 4)
    //=====================================================================
    E_PrimeSolventState.PS_Solvent4:

        IF NOT bPrimeRequired[4] THEN
            // Last solvent is not required → finish
            ePrimeState       := E_PrimeSolventState.PS_Completed;
            iStepCounter      := 0;
            bMovementComplete := FALSE;
        ELSE
            iActiveSolventPosition := 4;
            PrimeSolventCycle();

            IF bMovementComplete THEN
                ePrimeState       := E_PrimeSolventState.PS_Completed;
                iStepCounter      := 0;
                bMovementComplete := FALSE;
            END_IF
        END_IF


    //=====================================================================
    // COMPLETED
    //  - Terminal state of the prime sequence.
    //  - HMI is set to "Completed" and bDone is TRUE.
    //=====================================================================
    E_PrimeSolventState.PS_Completed:

        GVL_HMI.HMIAnimation.sLoadTextPrime  := 'Prime Completed';
        GVL_HMI.HMIAnimation.rLoadBarPrime   := 100.0;
        GVL_HMI.HMIAnimation.eIconStatePrime := E_IconState.Completed;

        bDone := TRUE;
        bBusy := FALSE;

END_CASE

ACTION BuildPrimeListFromRecipe:
(*
==============================================================================
 BuildPrimeListFromRecipe
------------------------------------------------------------------------------
 Purpose:
   - Inspect the active recipe and determine which solvents (1..4) are
     actually used in:
        * Rinse1
        * Rinse2
        * Wash1
        * Wash2
   - Build:
        bPrimeRequired[1..4]   → TRUE if solvent N is used in at least one step
        iNumSolventsToPrime    → number of unique solvents that must be primed
 Notes:
   - Recipe encoding:
        GVL_Recipe.stActiveRecipe.stSolventsTimes.aSolventN[1] = Rinse1 solvent
        GVL_Recipe.stActiveRecipe.stSolventsTimes.aSolventN[2] = Rinse2 solvent
        GVL_Recipe.stActiveRecipe.stSolventsTimes.aSolventN[3] = Wash1 solvent
        GVL_Recipe.stActiveRecipe.stSolventsTimes.aSolventN[4] = Wash2 solvent
   - Value 0 means "no solvent" / step disabled.
==============================================================================
*)

// Clear prime list and counter
FOR iSolventIdx := 1 TO 4 DO
    bPrimeRequired[iSolventIdx] := FALSE;
END_FOR;
iNumSolventsToPrime := 0;

// Scan recipe stages Rinse1..Wash2 (1..4)
FOR iStage := 1 TO 4 DO
    iSolventNum := GVL_Recipe.stActiveRecipe.stSolventsTimes.aSolventN[iStage];

    // Valid solvents are 1..4; 0 means "skip"
    IF (iSolventNum >= 1) AND (iSolventNum <= 4) THEN
        // Mark this solvent as required (idempotent)
        IF NOT bPrimeRequired[iSolventNum] THEN
            bPrimeRequired[iSolventNum] := TRUE;
        END_IF
    END_IF
END_FOR

// Count how many solvents will really be primed
FOR iSolventIdx := 1 TO 4 DO
    IF bPrimeRequired[iSolventIdx] THEN
        iNumSolventsToPrime := iNumSolventsToPrime + 1;
    END_IF
END_FOR
END_ACTION

